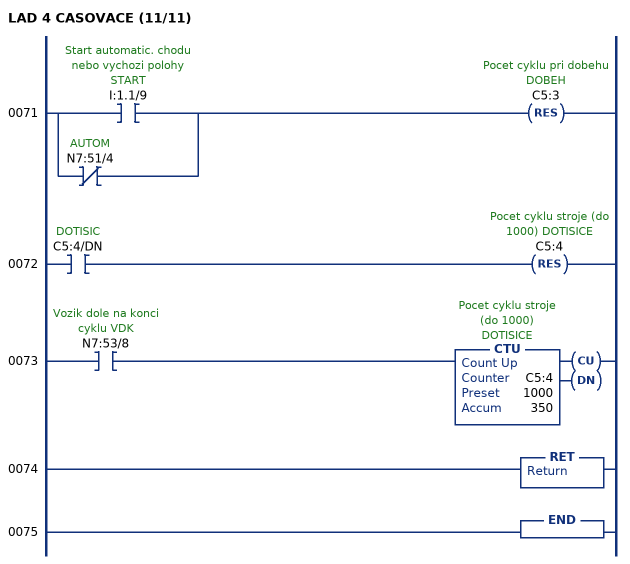
% Rung: 71 %
SOR BST XIC I:1.1/9 NXB XIO N7:51/4 BND RES C5:3 EOR
%   I:1.1/9  START  "Start automatic. chodu nebo vychozi polohy" %
%   N7:51/4  AUTOM %
%   C5:3  DOBEH  "Pocet cyklu pri dobehu" %
% Rung: 72 %
SOR XIC C5:4/DN RES C5:4 EOR
%   C5:4/DN  DOTISIC %
%   C5:4  DOTISICE  "Pocet cyklu stroje (do 1000)" %
% Rung: 73 %
SOR XIC N7:53/8 CTU C5:4 1000 350 EOR
%   N7:53/8  VDK  "Vozik dole na konci cyklu" %
%   C5:4  DOTISICE  "Pocet cyklu stroje (do 1000)" %
% Rung: 74 %
SOR RET EOR
% Rung: 75 %
SOR END EOR

LADDER 5 "DIAGN_SPOL"
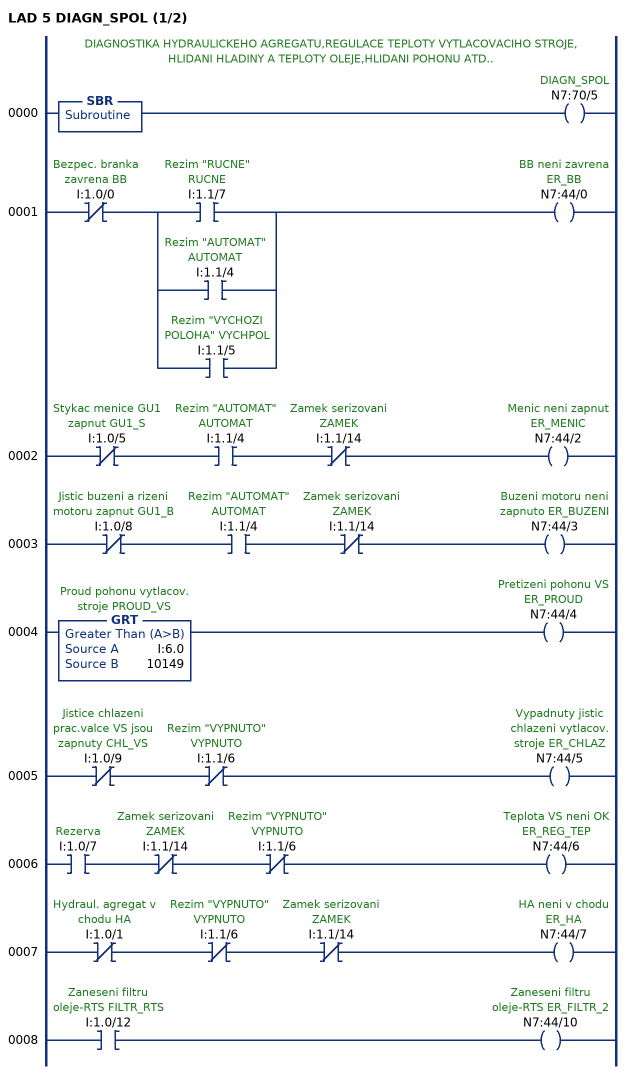
% Rung: 0 %
% DIAGNOSTIKA HYDRAULICKEHO AGREGATU,REGULACE TEPLOTY VYTLACOVACIHO STROJE,
% HLIDANI HLADINY A TEPLOTY OLEJE,HLIDANI POHONU ATD.. %
SOR SBR OTE N7:70/5 EOR
%   N7:70/5  DIAGN_SPOL %
% Rung: 1 %
SOR XIO I:1.0/0 BST XIC I:1.1/7 NXB XIC I:1.1/4 NXB XIC I:1.1/5 BND OTE N7:44/0 EOR
%   I:1.0/0  BB  "Bezpec. branka zavrena" %
%   I:1.1/7  RUCNE  "Rezim "RUCNE"" %
%   I:1.1/4  AUTOMAT  "Rezim "AUTOMAT"" %
%   I:1.1/5  VYCHPOL  "Rezim "VYCHOZI POLOHA"" %
%   N7:44/0  ER_BB  "BB neni zavrena" %
% Rung: 2 %
SOR XIO I:1.0/5 XIC I:1.1/4 XIO I:1.1/14 OTE N7:44/2 EOR
%   I:1.0/5  GU1_S  "Stykac menice GU1 zapnut" %
%   I:1.1/4  AUTOMAT  "Rezim "AUTOMAT"" %
%   I:1.1/14  ZAMEK  "Zamek serizovani" %
%   N7:44/2  ER_MENIC  "Menic neni zapnut" %
% Rung: 3 %
SOR XIO I:1.0/8 XIC I:1.1/4 XIO I:1.1/14 OTE N7:44/3 EOR
%   I:1.0/8  GU1_B  "Jistic buzeni a rizeni motoru zapnut" %
%   I:1.1/4  AUTOMAT  "Rezim "AUTOMAT"" %
%   I:1.1/14  ZAMEK  "Zamek serizovani" %
%   N7:44/3  ER_BUZENI  "Buzeni motoru neni zapnuto" %
% Rung: 4 %
SOR GRT I:6.0 10149 OTE N7:44/4 EOR
%   I:6.0  PROUD_VS  "Proud pohonu vytlacov. stroje" %
%   N7:44/4  ER_PROUD  "Pretizeni pohonu VS" %
% Rung: 5 %
SOR XIO I:1.0/9 XIO I:1.1/6 OTE N7:44/5 EOR
%   I:1.0/9  CHL_VS  "Jistice chlazeni prac.valce VS jsou zapnuty" %
%   I:1.1/6  VYPNUTO  "Rezim "VYPNUTO"" %
%   N7:44/5  ER_CHLAZ  "Vypadnuty jistic chlazeni vytlacov. stroje" %
% Rung: 6 %
SOR XIC I:1.0/7 XIO I:1.1/14 XIO I:1.1/6 OTE N7:44/6 EOR
%   I:1.0/7  "Rezerva" %
%   I:1.1/14  ZAMEK  "Zamek serizovani" %
%   I:1.1/6  VYPNUTO  "Rezim "VYPNUTO"" %
%   N7:44/6  ER_REG_TEP  "Teplota VS neni OK" %
% Rung: 7 %
SOR XIO I:1.0/1 XIO I:1.1/6 XIO I:1.1/14 OTE N7:44/7 EOR
%   I:1.0/1  HA  "Hydraul. agregat v chodu" %
%   I:1.1/6  VYPNUTO  "Rezim "VYPNUTO"" %
%   I:1.1/14  ZAMEK  "Zamek serizovani" %
%   N7:44/7  ER_HA  "HA neni v chodu" %
% Rung: 8 %
SOR XIC I:1.0/12 OTE N7:44/10 EOR
%   I:1.0/12  FILTR_RTS  "Zaneseni filtru oleje-RTS" %
%   N7:44/10  ER_FILTR_2  "Zaneseni filtru oleje-RTS" %

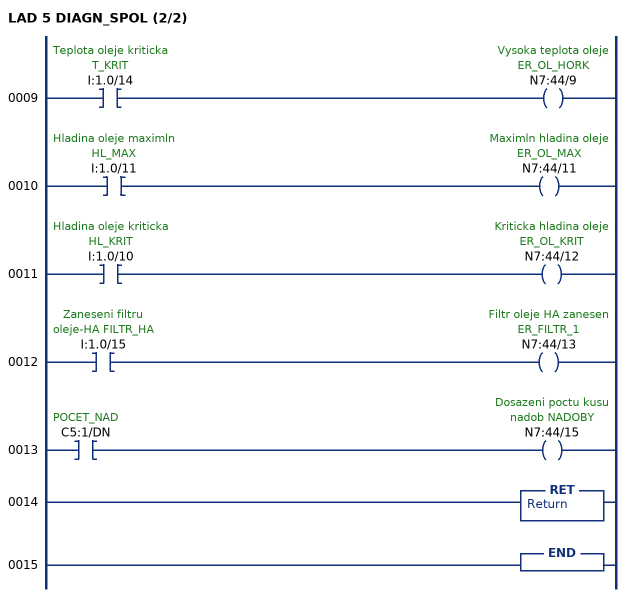
% Rung: 9 %
SOR XIC I:1.0/14 OTE N7:44/9 EOR
%   I:1.0/14  T_KRIT  "Teplota oleje kriticka" %
%   N7:44/9  ER_OL_HORK  "Vysoka teplota oleje" %
% Rung: 10 %
SOR XIC I:1.0/11 OTE N7:44/11 EOR
%   I:1.0/11  HL_MAX  "Hladina oleje maximln" %
%   N7:44/11  ER_OL_MAX  "Maximln hladina oleje" %
% Rung: 11 %
SOR XIC I:1.0/10 OTE N7:44/12 EOR
%   I:1.0/10  HL_KRIT  "Hladina oleje kriticka" %
%   N7:44/12  ER_OL_KRIT  "Kriticka hladina oleje" %
% Rung: 12 %
SOR XIC I:1.0/15 OTE N7:44/13 EOR
%   I:1.0/15  FILTR_HA  "Zaneseni filtru oleje-HA" %
%   N7:44/13  ER_FILTR_1  "Filtr oleje HA zanesen" %
% Rung: 13 %
SOR XIC C5:1/DN OTE N7:44/15 EOR
%   C5:1/DN  POCET_NAD %
%   N7:44/15  NADOBY  "Dosazeni poctu kusu nadob" %
% Rung: 14 %
SOR RET EOR
% Rung: 15 %
SOR END EOR

LADDER 6 "DIAGN_AUT"
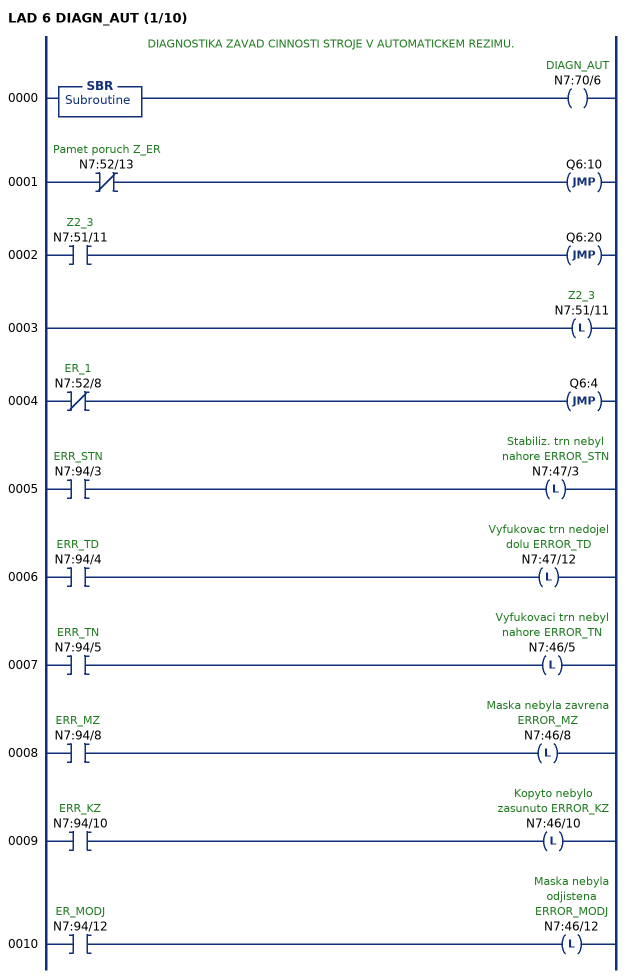
% Rung: 0 %
% DIAGNOSTIKA ZAVAD CINNOSTI STROJE V AUTOMATICKEM REZIMU. %
SOR SBR OTE N7:70/6 EOR
%   N7:70/6  DIAGN_AUT %
% Rung: 1 %
SOR XIO N7:52/13 JMP Q6:10 EOR
%   N7:52/13  Z_ER  "Pamet poruch" %
% Rung: 2 %
SOR XIC N7:51/11 JMP Q6:20 EOR
%   N7:51/11  Z2_3 %
% Rung: 3 %
SOR OTL N7:51/11 EOR
%   N7:51/11  Z2_3 %
% Rung: 4 %
SOR XIO N7:52/8 JMP Q6:4 EOR
%   N7:52/8  ER_1 %
% Rung: 5 %
SOR XIC N7:94/3 OTL N7:47/3 EOR
%   N7:94/3  ERR_STN %
%   N7:47/3  ERROR_STN  "Stabiliz. trn nebyl nahore" %
% Rung: 6 %
SOR XIC N7:94/4 OTL N7:47/12 EOR
%   N7:94/4  ERR_TD %
%   N7:47/12  ERROR_TD  "Vyfukovac trn nedojel dolu" %
% Rung: 7 %
SOR XIC N7:94/5 OTL N7:46/5 EOR
%   N7:94/5  ERR_TN %
%   N7:46/5  ERROR_TN  "Vyfukovaci trn nebyl nahore" %
% Rung: 8 %
SOR XIC N7:94/8 OTL N7:46/8 EOR
%   N7:94/8  ERR_MZ %
%   N7:46/8  ERROR_MZ  "Maska nebyla zavrena" %
% Rung: 9 %
SOR XIC N7:94/10 OTL N7:46/10 EOR
%   N7:94/10  ERR_KZ %
%   N7:46/10  ERROR_KZ  "Kopyto nebylo zasunuto" %
% Rung: 10 %
SOR XIC N7:94/12 OTL N7:46/12 EOR
%   N7:94/12  ER_MODJ %
%   N7:46/12  ERROR_MODJ  "Maska nebyla odjistena" %

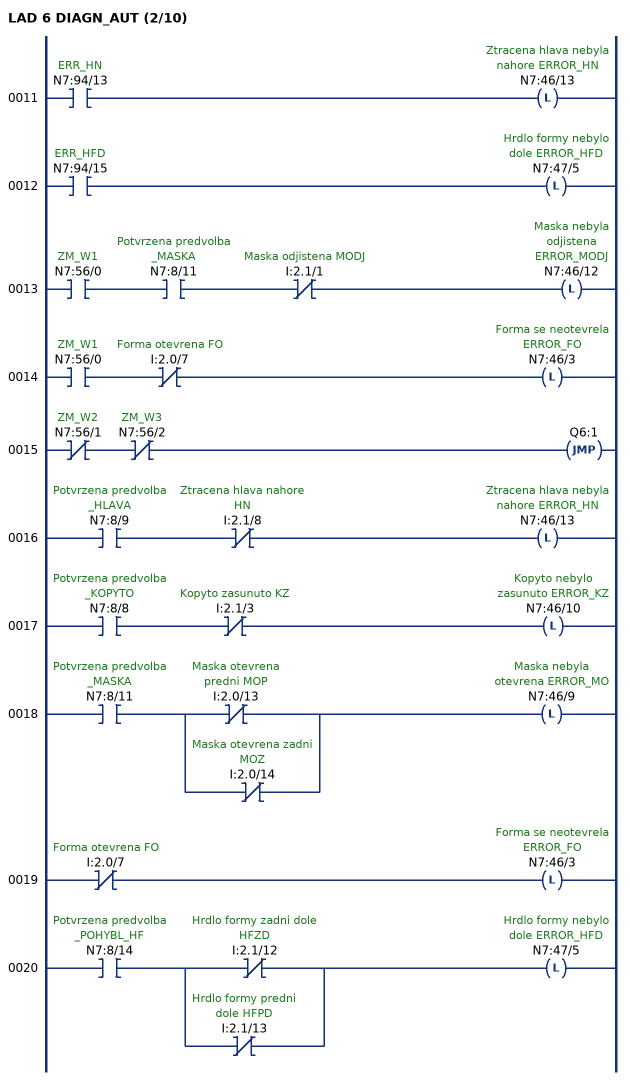
% Rung: 11 %
SOR XIC N7:94/13 OTL N7:46/13 EOR
%   N7:94/13  ERR_HN %
%   N7:46/13  ERROR_HN  "Ztracena hlava nebyla nahore" %
% Rung: 12 %
SOR XIC N7:94/15 OTL N7:47/5 EOR
%   N7:94/15  ERR_HFD %
%   N7:47/5  ERROR_HFD  "Hrdlo formy nebylo dole" %
% Rung: 13 %
SOR XIC N7:56/0 XIC N7:8/11 XIO I:2.1/1 OTL N7:46/12 EOR
%   N7:56/0  ZM_W1 %
%   N7:8/11  _MASKA  "Potvrzena predvolba" %
%   I:2.1/1  MODJ  "Maska odjistena" %
%   N7:46/12  ERROR_MODJ  "Maska nebyla odjistena" %
% Rung: 14 %
SOR XIC N7:56/0 XIO I:2.0/7 OTL N7:46/3 EOR
%   N7:56/0  ZM_W1 %
%   I:2.0/7  FO  "Forma otevrena" %
%   N7:46/3  ERROR_FO  "Forma se neotevrela" %
% Rung: 15 %
SOR XIO N7:56/1 XIO N7:56/2 JMP Q6:1 EOR
%   N7:56/1  ZM_W2 %
%   N7:56/2  ZM_W3 %
% Rung: 16 %
SOR XIC N7:8/9 XIO I:2.1/8 OTL N7:46/13 EOR
%   N7:8/9  _HLAVA  "Potvrzena predvolba" %
%   I:2.1/8  HN  "Ztracena hlava nahore" %
%   N7:46/13  ERROR_HN  "Ztracena hlava nebyla nahore" %
% Rung: 17 %
SOR XIC N7:8/8 XIO I:2.1/3 OTL N7:46/10 EOR
%   N7:8/8  _KOPYTO  "Potvrzena predvolba" %
%   I:2.1/3  KZ  "Kopyto zasunuto" %
%   N7:46/10  ERROR_KZ  "Kopyto nebylo zasunuto" %
% Rung: 18 %
SOR XIC N7:8/11 BST XIO I:2.0/13 NXB XIO I:2.0/14 BND OTL N7:46/9 EOR
%   N7:8/11  _MASKA  "Potvrzena predvolba" %
%   I:2.0/13  MOP  "Maska otevrena predni" %
%   I:2.0/14  MOZ  "Maska otevrena zadni" %
%   N7:46/9  ERROR_MO  "Maska nebyla otevrena" %
% Rung: 19 %
SOR XIO I:2.0/7 OTL N7:46/3 EOR
%   I:2.0/7  FO  "Forma otevrena" %
%   N7:46/3  ERROR_FO  "Forma se neotevrela" %
% Rung: 20 %
SOR XIC N7:8/14 BST XIO I:2.1/12 NXB XIO I:2.1/13 BND OTL N7:47/5 EOR
%   N7:8/14  _POHYBL_HF  "Potvrzena predvolba" %
%   I:2.1/12  HFZD  "Hrdlo formy zadni dole" %
%   I:2.1/13  HFPD  "Hrdlo formy predni dole" %
%   N7:47/5  ERROR_HFD  "Hrdlo formy nebylo dole" %

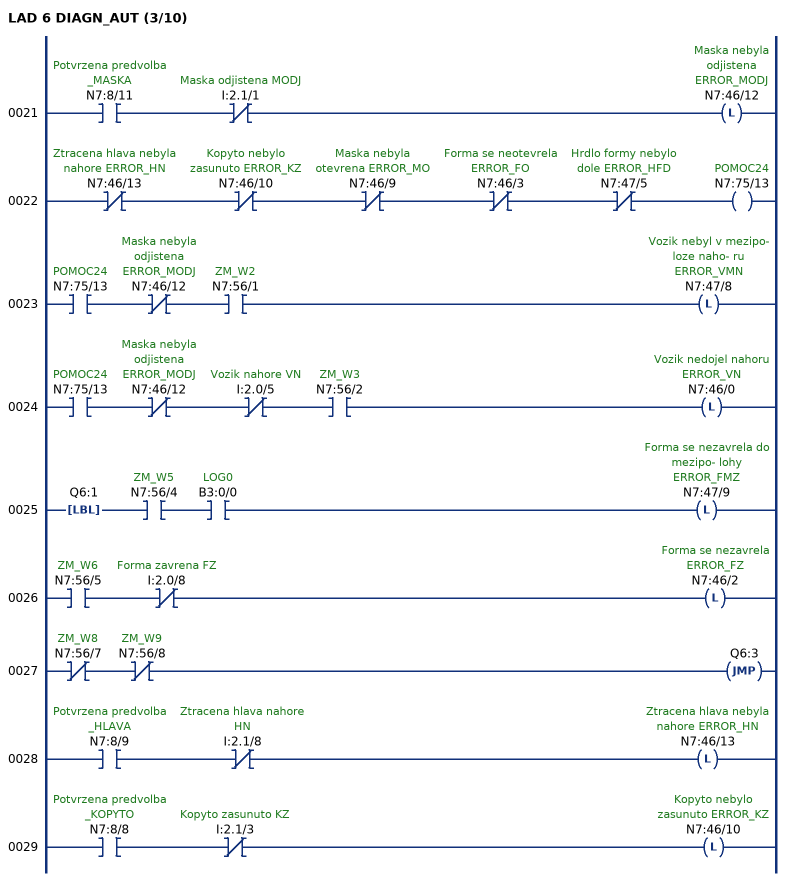
% Rung: 21 %
SOR XIC N7:8/11 XIO I:2.1/1 OTL N7:46/12 EOR
%   N7:8/11  _MASKA  "Potvrzena predvolba" %
%   I:2.1/1  MODJ  "Maska odjistena" %
%   N7:46/12  ERROR_MODJ  "Maska nebyla odjistena" %
% Rung: 22 %
SOR XIO N7:46/13 XIO N7:46/10 XIO N7:46/9 XIO N7:46/3 XIO N7:47/5 OTE N7:75/13 EOR
%   N7:46/13  ERROR_HN  "Ztracena hlava nebyla nahore" %
%   N7:46/10  ERROR_KZ  "Kopyto nebylo zasunuto" %
%   N7:46/9  ERROR_MO  "Maska nebyla otevrena" %
%   N7:46/3  ERROR_FO  "Forma se neotevrela" %
%   N7:47/5  ERROR_HFD  "Hrdlo formy nebylo dole" %
%   N7:75/13  POMOC24 %
% Rung: 23 %
SOR XIC N7:75/13 XIO N7:46/12 XIC N7:56/1 OTL N7:47/8 EOR
%   N7:75/13  POMOC24 %
%   N7:46/12  ERROR_MODJ  "Maska nebyla odjistena" %
%   N7:56/1  ZM_W2 %
%   N7:47/8  ERROR_VMN  "Vozik nebyl v mezipo- loze naho- ru" %
% Rung: 24 %
SOR XIC N7:75/13 XIO N7:46/12 XIO I:2.0/5 XIC N7:56/2 OTL N7:46/0 EOR
%   N7:75/13  POMOC24 %
%   N7:46/12  ERROR_MODJ  "Maska nebyla odjistena" %
%   I:2.0/5  VN  "Vozik nahore" %
%   N7:56/2  ZM_W3 %
%   N7:46/0  ERROR_VN  "Vozik nedojel nahoru" %
% Rung: 25 %
SOR LBL Q6:1 XIC N7:56/4 XIC B3:0/0 OTL N7:47/9 EOR
%   N7:56/4  ZM_W5 %
%   B3:0/0  LOG0 %
%   N7:47/9  ERROR_FMZ  "Forma se nezavrela do mezipo- lohy" %
% Rung: 26 %
SOR XIC N7:56/5 XIO I:2.0/8 OTL N7:46/2 EOR
%   N7:56/5  ZM_W6 %
%   I:2.0/8  FZ  "Forma zavrena" %
%   N7:46/2  ERROR_FZ  "Forma se nezavrela" %
% Rung: 27 %
SOR XIO N7:56/7 XIO N7:56/8 JMP Q6:3 EOR
%   N7:56/7  ZM_W8 %
%   N7:56/8  ZM_W9 %
% Rung: 28 %
SOR XIC N7:8/9 XIO I:2.1/8 OTL N7:46/13 EOR
%   N7:8/9  _HLAVA  "Potvrzena predvolba" %
%   I:2.1/8  HN  "Ztracena hlava nahore" %
%   N7:46/13  ERROR_HN  "Ztracena hlava nebyla nahore" %
% Rung: 29 %
SOR XIC N7:8/8 XIO I:2.1/3 OTL N7:46/10 EOR
%   N7:8/8  _KOPYTO  "Potvrzena predvolba" %
%   I:2.1/3  KZ  "Kopyto zasunuto" %
%   N7:46/10  ERROR_KZ  "Kopyto nebylo zasunuto" %

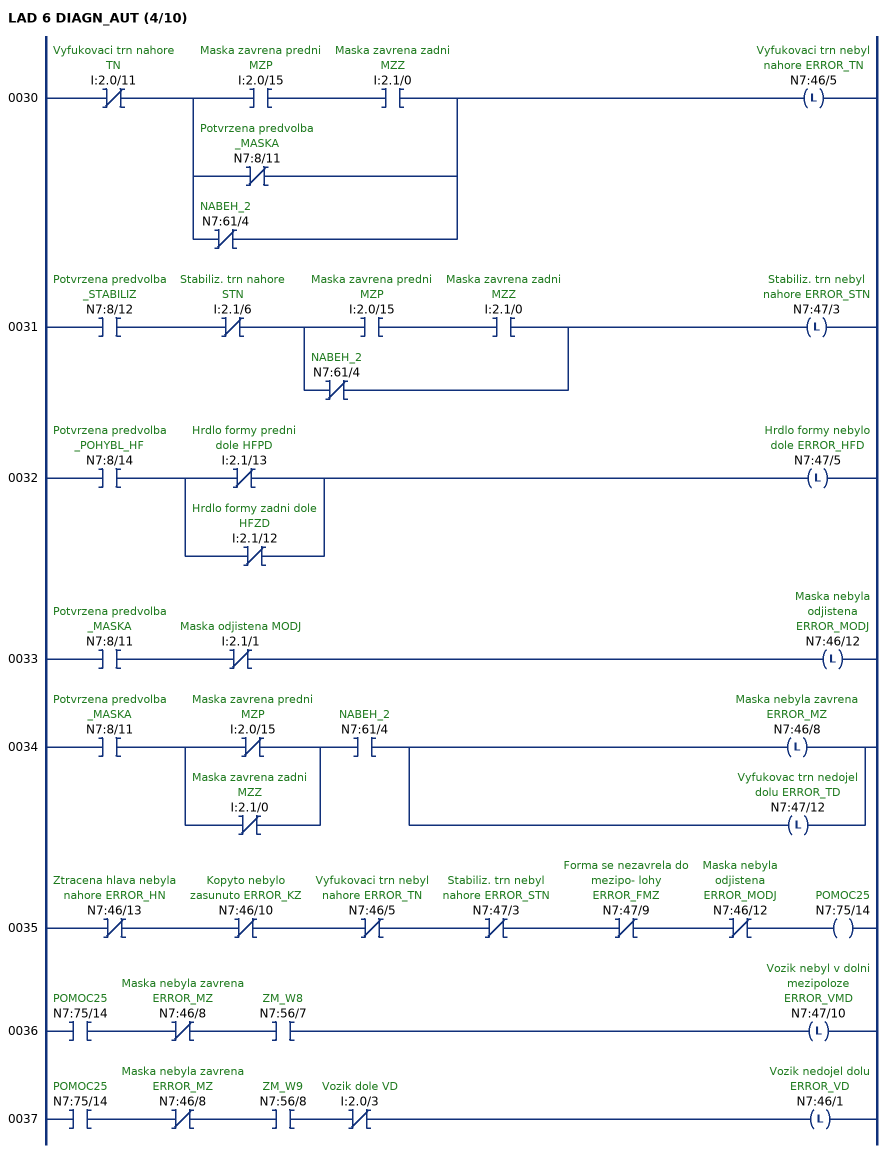
% Rung: 30 %
SOR XIO I:2.0/11 BST XIC I:2.0/15 XIC I:2.1/0 NXB XIO N7:8/11 NXB XIO N7:61/4 BND OTL N7:46/5 EOR
%   I:2.0/11  TN  "Vyfukovaci trn nahore" %
%   I:2.0/15  MZP  "Maska zavrena predni" %
%   I:2.1/0  MZZ  "Maska zavrena zadni" %
%   N7:8/11  _MASKA  "Potvrzena predvolba" %
%   N7:61/4  NABEH_2 %
%   N7:46/5  ERROR_TN  "Vyfukovaci trn nebyl nahore" %
% Rung: 31 %
SOR XIC N7:8/12 XIO I:2.1/6 BST XIC I:2.0/15 XIC I:2.1/0 NXB XIO N7:61/4 BND OTL N7:47/3 EOR
%   N7:8/12  _STABILIZ  "Potvrzena predvolba" %
%   I:2.1/6  STN  "Stabiliz. trn nahore" %
%   I:2.0/15  MZP  "Maska zavrena predni" %
%   I:2.1/0  MZZ  "Maska zavrena zadni" %
%   N7:61/4  NABEH_2 %
%   N7:47/3  ERROR_STN  "Stabiliz. trn nebyl nahore" %
% Rung: 32 %
SOR XIC N7:8/14 BST XIO I:2.1/13 NXB XIO I:2.1/12 BND OTL N7:47/5 EOR
%   N7:8/14  _POHYBL_HF  "Potvrzena predvolba" %
%   I:2.1/13  HFPD  "Hrdlo formy predni dole" %
%   I:2.1/12  HFZD  "Hrdlo formy zadni dole" %
%   N7:47/5  ERROR_HFD  "Hrdlo formy nebylo dole" %
% Rung: 33 %
SOR XIC N7:8/11 XIO I:2.1/1 OTL N7:46/12 EOR
%   N7:8/11  _MASKA  "Potvrzena predvolba" %
%   I:2.1/1  MODJ  "Maska odjistena" %
%   N7:46/12  ERROR_MODJ  "Maska nebyla odjistena" %
% Rung: 34 %
SOR XIC N7:8/11 BST XIO I:2.0/15 NXB XIO I:2.1/0 BND XIC N7:61/4 BST OTL N7:46/8 NXB OTL N7:47/12 BND EOR
%   N7:8/11  _MASKA  "Potvrzena predvolba" %
%   I:2.0/15  MZP  "Maska zavrena predni" %
%   I:2.1/0  MZZ  "Maska zavrena zadni" %
%   N7:61/4  NABEH_2 %
%   N7:46/8  ERROR_MZ  "Maska nebyla zavrena" %
%   N7:47/12  ERROR_TD  "Vyfukovac trn nedojel dolu" %
% Rung: 35 %
SOR XIO N7:46/13 XIO N7:46/10 XIO N7:46/5 XIO N7:47/3 XIO N7:47/9 XIO N7:46/12 OTE N7:75/14 EOR
%   N7:46/13  ERROR_HN  "Ztracena hlava nebyla nahore" %
%   N7:46/10  ERROR_KZ  "Kopyto nebylo zasunuto" %
%   N7:46/5  ERROR_TN  "Vyfukovaci trn nebyl nahore" %
%   N7:47/3  ERROR_STN  "Stabiliz. trn nebyl nahore" %
%   N7:47/9  ERROR_FMZ  "Forma se nezavrela do mezipo- lohy" %
%   N7:46/12  ERROR_MODJ  "Maska nebyla odjistena" %
%   N7:75/14  POMOC25 %
% Rung: 36 %
SOR XIC N7:75/14 XIO N7:46/8 XIC N7:56/7 OTL N7:47/10 EOR
%   N7:75/14  POMOC25 %
%   N7:46/8  ERROR_MZ  "Maska nebyla zavrena" %
%   N7:56/7  ZM_W8 %
%   N7:47/10  ERROR_VMD  "Vozik nebyl v dolni mezipoloze" %
% Rung: 37 %
SOR XIC N7:75/14 XIO N7:46/8 XIC N7:56/8 XIO I:2.0/3 OTL N7:46/1 EOR
%   N7:75/14  POMOC25 %
%   N7:46/8  ERROR_MZ  "Maska nebyla zavrena" %
%   N7:56/8  ZM_W9 %
%   I:2.0/3  VD  "Vozik dole" %
%   N7:46/1  ERROR_VD  "Vozik nedojel dolu" %

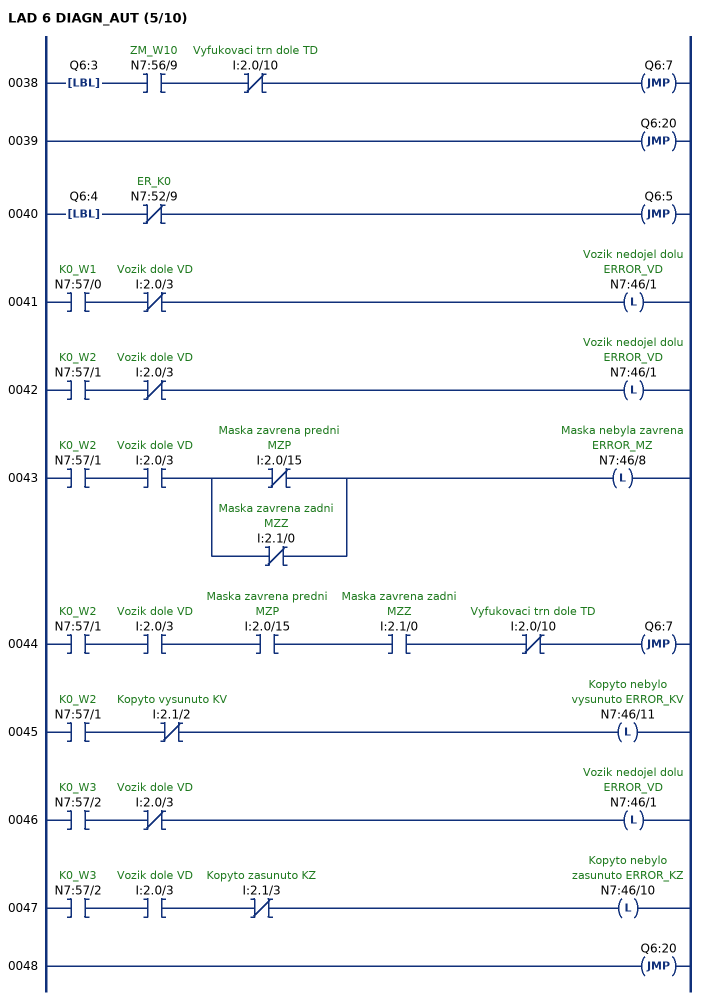
% Rung: 38 %
SOR LBL Q6:3 XIC N7:56/9 XIO I:2.0/10 JMP Q6:7 EOR
%   N7:56/9  ZM_W10 %
%   I:2.0/10  TD  "Vyfukovaci trn dole" %
% Rung: 39 %
SOR JMP Q6:20 EOR
% Rung: 40 %
SOR LBL Q6:4 XIO N7:52/9 JMP Q6:5 EOR
%   N7:52/9  ER_K0 %
% Rung: 41 %
SOR XIC N7:57/0 XIO I:2.0/3 OTL N7:46/1 EOR
%   N7:57/0  K0_W1 %
%   I:2.0/3  VD  "Vozik dole" %
%   N7:46/1  ERROR_VD  "Vozik nedojel dolu" %
% Rung: 42 %
SOR XIC N7:57/1 XIO I:2.0/3 OTL N7:46/1 EOR
%   N7:57/1  K0_W2 %
%   I:2.0/3  VD  "Vozik dole" %
%   N7:46/1  ERROR_VD  "Vozik nedojel dolu" %
% Rung: 43 %
SOR XIC N7:57/1 XIC I:2.0/3 BST XIO I:2.0/15 NXB XIO I:2.1/0 BND OTL N7:46/8 EOR
%   N7:57/1  K0_W2 %
%   I:2.0/3  VD  "Vozik dole" %
%   I:2.0/15  MZP  "Maska zavrena predni" %
%   I:2.1/0  MZZ  "Maska zavrena zadni" %
%   N7:46/8  ERROR_MZ  "Maska nebyla zavrena" %
% Rung: 44 %
SOR XIC N7:57/1 XIC I:2.0/3 XIC I:2.0/15 XIC I:2.1/0 XIO I:2.0/10 JMP Q6:7 EOR
%   N7:57/1  K0_W2 %
%   I:2.0/3  VD  "Vozik dole" %
%   I:2.0/15  MZP  "Maska zavrena predni" %
%   I:2.1/0  MZZ  "Maska zavrena zadni" %
%   I:2.0/10  TD  "Vyfukovaci trn dole" %
% Rung: 45 %
SOR XIC N7:57/1 XIO I:2.1/2 OTL N7:46/11 EOR
%   N7:57/1  K0_W2 %
%   I:2.1/2  KV  "Kopyto vysunuto" %
%   N7:46/11  ERROR_KV  "Kopyto nebylo vysunuto" %
% Rung: 46 %
SOR XIC N7:57/2 XIO I:2.0/3 OTL N7:46/1 EOR
%   N7:57/2  K0_W3 %
%   I:2.0/3  VD  "Vozik dole" %
%   N7:46/1  ERROR_VD  "Vozik nedojel dolu" %
% Rung: 47 %
SOR XIC N7:57/2 XIC I:2.0/3 XIO I:2.1/3 OTL N7:46/10 EOR
%   N7:57/2  K0_W3 %
%   I:2.0/3  VD  "Vozik dole" %
%   I:2.1/3  KZ  "Kopyto zasunuto" %
%   N7:46/10  ERROR_KZ  "Kopyto nebylo zasunuto" %
% Rung: 48 %
SOR JMP Q6:20 EOR

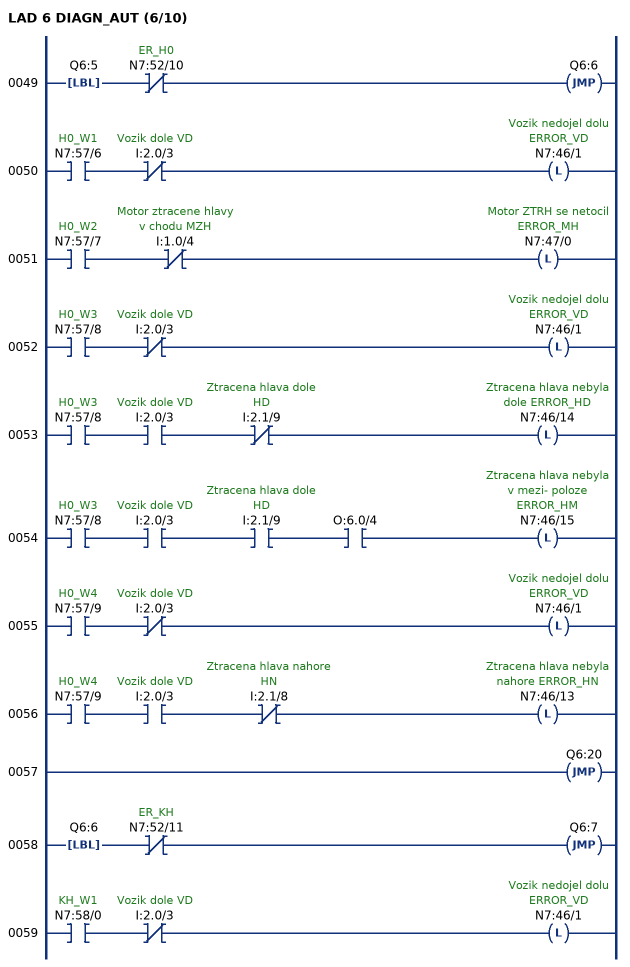
% Rung: 49 %
SOR LBL Q6:5 XIO N7:52/10 JMP Q6:6 EOR
%   N7:52/10  ER_H0 %
% Rung: 50 %
SOR XIC N7:57/6 XIO I:2.0/3 OTL N7:46/1 EOR
%   N7:57/6  H0_W1 %
%   I:2.0/3  VD  "Vozik dole" %
%   N7:46/1  ERROR_VD  "Vozik nedojel dolu" %
% Rung: 51 %
SOR XIC N7:57/7 XIO I:1.0/4 OTL N7:47/0 EOR
%   N7:57/7  H0_W2 %
%   I:1.0/4  MZH  "Motor ztracene hlavy v chodu" %
%   N7:47/0  ERROR_MH  "Motor ZTRH se netocil" %
% Rung: 52 %
SOR XIC N7:57/8 XIO I:2.0/3 OTL N7:46/1 EOR
%   N7:57/8  H0_W3 %
%   I:2.0/3  VD  "Vozik dole" %
%   N7:46/1  ERROR_VD  "Vozik nedojel dolu" %
% Rung: 53 %
SOR XIC N7:57/8 XIC I:2.0/3 XIO I:2.1/9 OTL N7:46/14 EOR
%   N7:57/8  H0_W3 %
%   I:2.0/3  VD  "Vozik dole" %
%   I:2.1/9  HD  "Ztracena hlava dole" %
%   N7:46/14  ERROR_HD  "Ztracena hlava nebyla dole" %
% Rung: 54 %
SOR XIC N7:57/8 XIC I:2.0/3 XIC I:2.1/9 XIC O:6.0/4 OTL N7:46/15 EOR
%   N7:57/8  H0_W3 %
%   I:2.0/3  VD  "Vozik dole" %
%   I:2.1/9  HD  "Ztracena hlava dole" %
%   N7:46/15  ERROR_HM  "Ztracena hlava nebyla v mezi- poloze" %
% Rung: 55 %
SOR XIC N7:57/9 XIO I:2.0/3 OTL N7:46/1 EOR
%   N7:57/9  H0_W4 %
%   I:2.0/3  VD  "Vozik dole" %
%   N7:46/1  ERROR_VD  "Vozik nedojel dolu" %
% Rung: 56 %
SOR XIC N7:57/9 XIC I:2.0/3 XIO I:2.1/8 OTL N7:46/13 EOR
%   N7:57/9  H0_W4 %
%   I:2.0/3  VD  "Vozik dole" %
%   I:2.1/8  HN  "Ztracena hlava nahore" %
%   N7:46/13  ERROR_HN  "Ztracena hlava nebyla nahore" %
% Rung: 57 %
SOR JMP Q6:20 EOR
% Rung: 58 %
SOR LBL Q6:6 XIO N7:52/11 JMP Q6:7 EOR
%   N7:52/11  ER_KH %
% Rung: 59 %
SOR XIC N7:58/0 XIO I:2.0/3 OTL N7:46/1 EOR
%   N7:58/0  KH_W1 %
%   I:2.0/3  VD  "Vozik dole" %
%   N7:46/1  ERROR_VD  "Vozik nedojel dolu" %

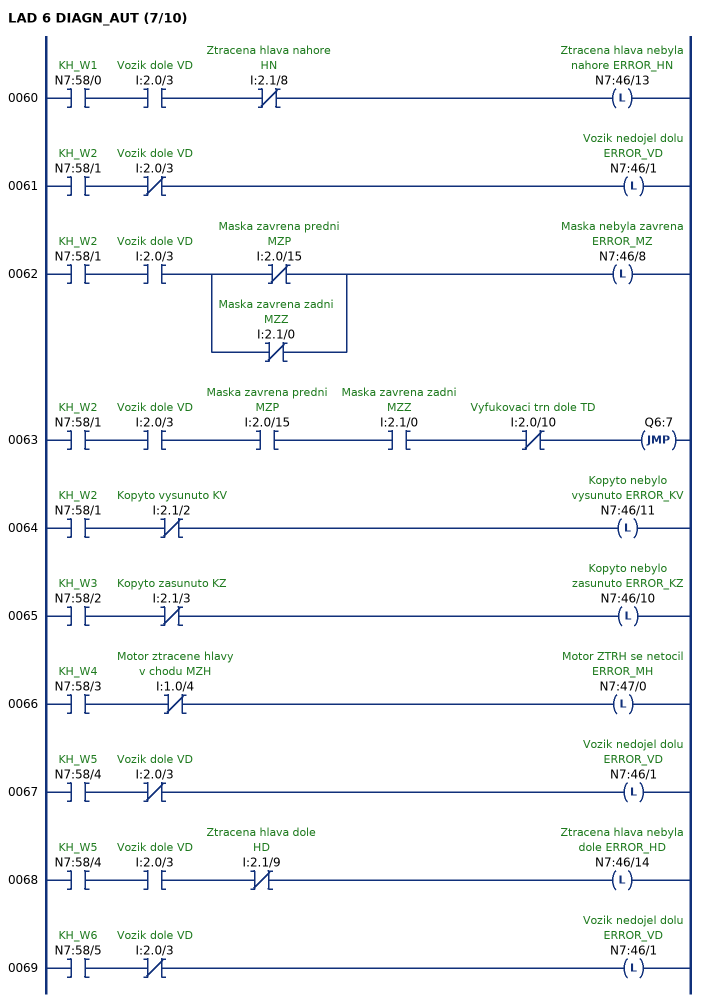
% Rung: 60 %
SOR XIC N7:58/0 XIC I:2.0/3 XIO I:2.1/8 OTL N7:46/13 EOR
%   N7:58/0  KH_W1 %
%   I:2.0/3  VD  "Vozik dole" %
%   I:2.1/8  HN  "Ztracena hlava nahore" %
%   N7:46/13  ERROR_HN  "Ztracena hlava nebyla nahore" %
% Rung: 61 %
SOR XIC N7:58/1 XIO I:2.0/3 OTL N7:46/1 EOR
%   N7:58/1  KH_W2 %
%   I:2.0/3  VD  "Vozik dole" %
%   N7:46/1  ERROR_VD  "Vozik nedojel dolu" %
% Rung: 62 %
SOR XIC N7:58/1 XIC I:2.0/3 BST XIO I:2.0/15 NXB XIO I:2.1/0 BND OTL N7:46/8 EOR
%   N7:58/1  KH_W2 %
%   I:2.0/3  VD  "Vozik dole" %
%   I:2.0/15  MZP  "Maska zavrena predni" %
%   I:2.1/0  MZZ  "Maska zavrena zadni" %
%   N7:46/8  ERROR_MZ  "Maska nebyla zavrena" %
% Rung: 63 %
SOR XIC N7:58/1 XIC I:2.0/3 XIC I:2.0/15 XIC I:2.1/0 XIO I:2.0/10 JMP Q6:7 EOR
%   N7:58/1  KH_W2 %
%   I:2.0/3  VD  "Vozik dole" %
%   I:2.0/15  MZP  "Maska zavrena predni" %
%   I:2.1/0  MZZ  "Maska zavrena zadni" %
%   I:2.0/10  TD  "Vyfukovaci trn dole" %
% Rung: 64 %
SOR XIC N7:58/1 XIO I:2.1/2 OTL N7:46/11 EOR
%   N7:58/1  KH_W2 %
%   I:2.1/2  KV  "Kopyto vysunuto" %
%   N7:46/11  ERROR_KV  "Kopyto nebylo vysunuto" %
% Rung: 65 %
SOR XIC N7:58/2 XIO I:2.1/3 OTL N7:46/10 EOR
%   N7:58/2  KH_W3 %
%   I:2.1/3  KZ  "Kopyto zasunuto" %
%   N7:46/10  ERROR_KZ  "Kopyto nebylo zasunuto" %
% Rung: 66 %
SOR XIC N7:58/3 XIO I:1.0/4 OTL N7:47/0 EOR
%   N7:58/3  KH_W4 %
%   I:1.0/4  MZH  "Motor ztracene hlavy v chodu" %
%   N7:47/0  ERROR_MH  "Motor ZTRH se netocil" %
% Rung: 67 %
SOR XIC N7:58/4 XIO I:2.0/3 OTL N7:46/1 EOR
%   N7:58/4  KH_W5 %
%   I:2.0/3  VD  "Vozik dole" %
%   N7:46/1  ERROR_VD  "Vozik nedojel dolu" %
% Rung: 68 %
SOR XIC N7:58/4 XIC I:2.0/3 XIO I:2.1/9 OTL N7:46/14 EOR
%   N7:58/4  KH_W5 %
%   I:2.0/3  VD  "Vozik dole" %
%   I:2.1/9  HD  "Ztracena hlava dole" %
%   N7:46/14  ERROR_HD  "Ztracena hlava nebyla dole" %
% Rung: 69 %
SOR XIC N7:58/5 XIO I:2.0/3 OTL N7:46/1 EOR
%   N7:58/5  KH_W6 %
%   I:2.0/3  VD  "Vozik dole" %
%   N7:46/1  ERROR_VD  "Vozik nedojel dolu" %

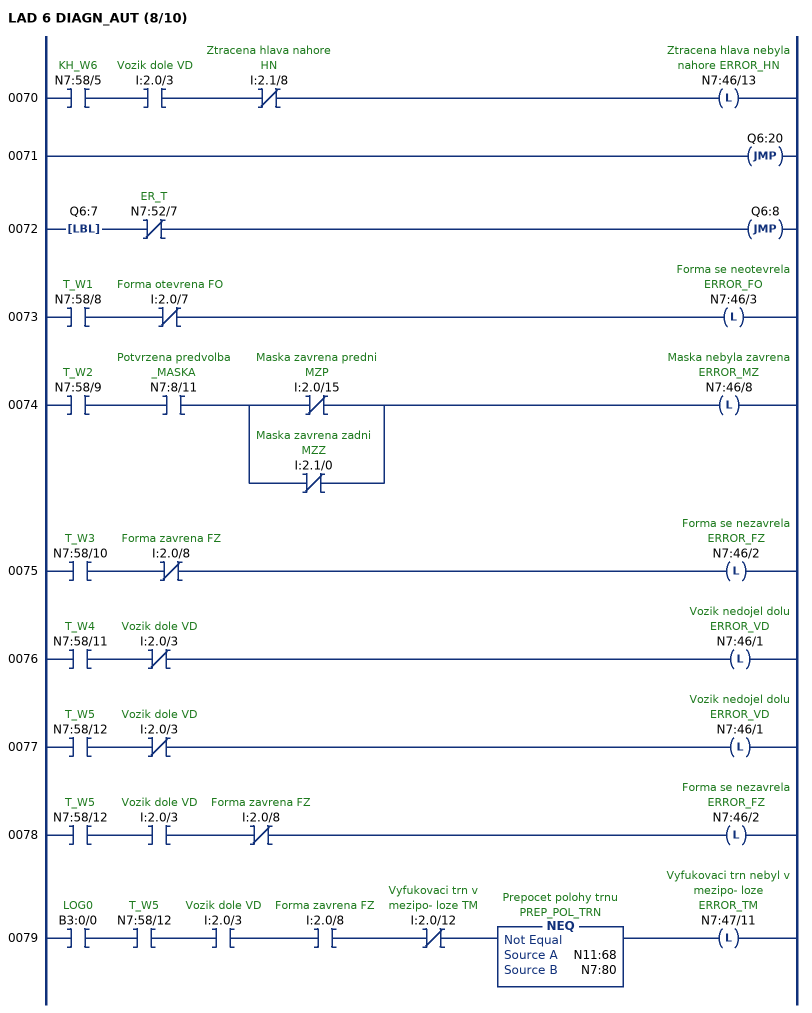
% Rung: 70 %
SOR XIC N7:58/5 XIC I:2.0/3 XIO I:2.1/8 OTL N7:46/13 EOR
%   N7:58/5  KH_W6 %
%   I:2.0/3  VD  "Vozik dole" %
%   I:2.1/8  HN  "Ztracena hlava nahore" %
%   N7:46/13  ERROR_HN  "Ztracena hlava nebyla nahore" %
% Rung: 71 %
SOR JMP Q6:20 EOR
% Rung: 72 %
SOR LBL Q6:7 XIO N7:52/7 JMP Q6:8 EOR
%   N7:52/7  ER_T %
% Rung: 73 %
SOR XIC N7:58/8 XIO I:2.0/7 OTL N7:46/3 EOR
%   N7:58/8  T_W1 %
%   I:2.0/7  FO  "Forma otevrena" %
%   N7:46/3  ERROR_FO  "Forma se neotevrela" %
% Rung: 74 %
SOR XIC N7:58/9 XIC N7:8/11 BST XIO I:2.0/15 NXB XIO I:2.1/0 BND OTL N7:46/8 EOR
%   N7:58/9  T_W2 %
%   N7:8/11  _MASKA  "Potvrzena predvolba" %
%   I:2.0/15  MZP  "Maska zavrena predni" %
%   I:2.1/0  MZZ  "Maska zavrena zadni" %
%   N7:46/8  ERROR_MZ  "Maska nebyla zavrena" %
% Rung: 75 %
SOR XIC N7:58/10 XIO I:2.0/8 OTL N7:46/2 EOR
%   N7:58/10  T_W3 %
%   I:2.0/8  FZ  "Forma zavrena" %
%   N7:46/2  ERROR_FZ  "Forma se nezavrela" %
% Rung: 76 %
SOR XIC N7:58/11 XIO I:2.0/3 OTL N7:46/1 EOR
%   N7:58/11  T_W4 %
%   I:2.0/3  VD  "Vozik dole" %
%   N7:46/1  ERROR_VD  "Vozik nedojel dolu" %
% Rung: 77 %
SOR XIC N7:58/12 XIO I:2.0/3 OTL N7:46/1 EOR
%   N7:58/12  T_W5 %
%   I:2.0/3  VD  "Vozik dole" %
%   N7:46/1  ERROR_VD  "Vozik nedojel dolu" %
% Rung: 78 %
SOR XIC N7:58/12 XIC I:2.0/3 XIO I:2.0/8 OTL N7:46/2 EOR
%   N7:58/12  T_W5 %
%   I:2.0/3  VD  "Vozik dole" %
%   I:2.0/8  FZ  "Forma zavrena" %
%   N7:46/2  ERROR_FZ  "Forma se nezavrela" %
% Rung: 79 %
SOR XIC B3:0/0 XIC N7:58/12 XIC I:2.0/3 XIC I:2.0/8 XIO I:2.0/12 NEQ N11:68 N7:80 OTL N7:47/11 EOR
%   B3:0/0  LOG0 %
%   N7:58/12  T_W5 %
%   I:2.0/3  VD  "Vozik dole" %
%   I:2.0/8  FZ  "Forma zavrena" %
%   I:2.0/12  TM  "Vyfukovaci trn v mezipo- loze" %
%   N11:68  PREP_POL_TRN  "Prepocet polohy trnu" %
%   N7:47/11  ERROR_TM  "Vyfukovaci trn nebyl v mezipo- loze" %

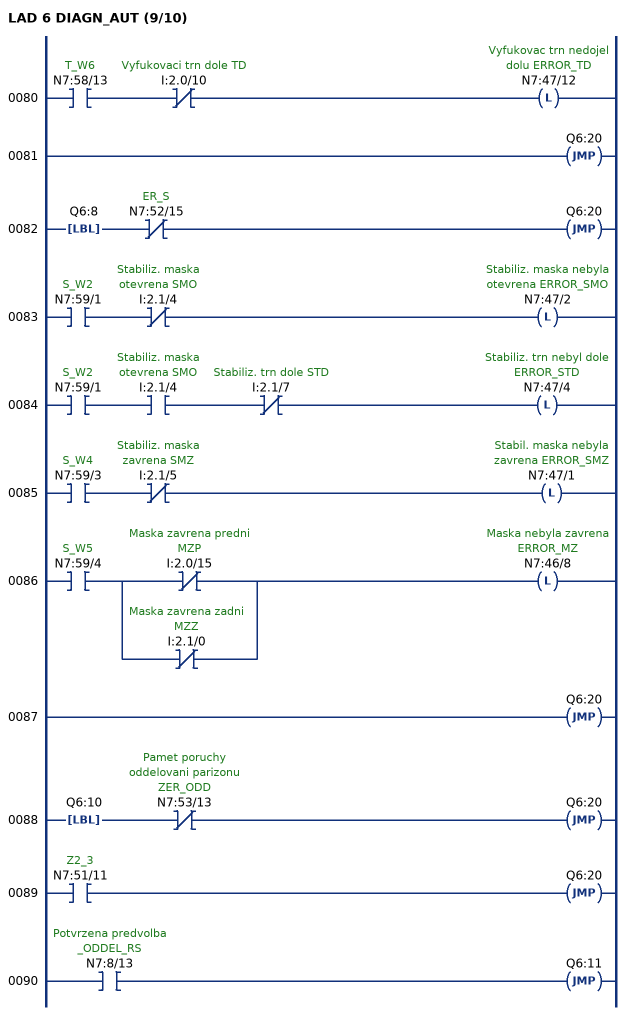
% Rung: 80 %
SOR XIC N7:58/13 XIO I:2.0/10 OTL N7:47/12 EOR
%   N7:58/13  T_W6 %
%   I:2.0/10  TD  "Vyfukovaci trn dole" %
%   N7:47/12  ERROR_TD  "Vyfukovac trn nedojel dolu" %
% Rung: 81 %
SOR JMP Q6:20 EOR
% Rung: 82 %
SOR LBL Q6:8 XIO N7:52/15 JMP Q6:20 EOR
%   N7:52/15  ER_S %
% Rung: 83 %
SOR XIC N7:59/1 XIO I:2.1/4 OTL N7:47/2 EOR
%   N7:59/1  S_W2 %
%   I:2.1/4  SMO  "Stabiliz. maska otevrena" %
%   N7:47/2  ERROR_SMO  "Stabiliz. maska nebyla otevrena" %
% Rung: 84 %
SOR XIC N7:59/1 XIC I:2.1/4 XIO I:2.1/7 OTL N7:47/4 EOR
%   N7:59/1  S_W2 %
%   I:2.1/4  SMO  "Stabiliz. maska otevrena" %
%   I:2.1/7  STD  "Stabiliz. trn dole" %
%   N7:47/4  ERROR_STD  "Stabiliz. trn nebyl dole" %
% Rung: 85 %
SOR XIC N7:59/3 XIO I:2.1/5 OTL N7:47/1 EOR
%   N7:59/3  S_W4 %
%   I:2.1/5  SMZ  "Stabiliz. maska zavrena" %
%   N7:47/1  ERROR_SMZ  "Stabil. maska nebyla zavrena" %
% Rung: 86 %
SOR XIC N7:59/4 BST XIO I:2.0/15 NXB XIO I:2.1/0 BND OTL N7:46/8 EOR
%   N7:59/4  S_W5 %
%   I:2.0/15  MZP  "Maska zavrena predni" %
%   I:2.1/0  MZZ  "Maska zavrena zadni" %
%   N7:46/8  ERROR_MZ  "Maska nebyla zavrena" %
% Rung: 87 %
SOR JMP Q6:20 EOR
% Rung: 88 %
SOR LBL Q6:10 XIO N7:53/13 JMP Q6:20 EOR
%   N7:53/13  ZER_ODD  "Pamet poruchy oddelovani parizonu" %
% Rung: 89 %
SOR XIC N7:51/11 JMP Q6:20 EOR
%   N7:51/11  Z2_3 %
% Rung: 90 %
SOR XIC N7:8/13 JMP Q6:11 EOR
%   N7:8/13  _ODDEL_RS  "Potvrzena predvolba" %

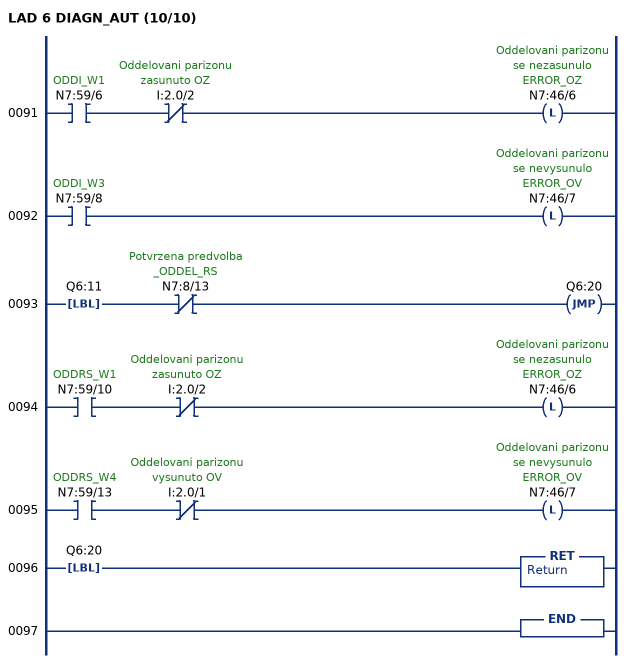
% Rung: 91 %
SOR XIC N7:59/6 XIO I:2.0/2 OTL N7:46/6 EOR
%   N7:59/6  ODDI_W1 %
%   I:2.0/2  OZ  "Oddelovani parizonu zasunuto" %
%   N7:46/6  ERROR_OZ  "Oddelovani parizonu se nezasunulo" %
% Rung: 92 %
SOR XIC N7:59/8 OTL N7:46/7 EOR
%   N7:59/8  ODDI_W3 %
%   N7:46/7  ERROR_OV  "Oddelovani parizonu se nevysunulo" %
% Rung: 93 %
SOR LBL Q6:11 XIO N7:8/13 JMP Q6:20 EOR
%   N7:8/13  _ODDEL_RS  "Potvrzena predvolba" %
% Rung: 94 %
SOR XIC N7:59/10 XIO I:2.0/2 OTL N7:46/6 EOR
%   N7:59/10  ODDRS_W1 %
%   I:2.0/2  OZ  "Oddelovani parizonu zasunuto" %
%   N7:46/6  ERROR_OZ  "Oddelovani parizonu se nezasunulo" %
% Rung: 95 %
SOR XIC N7:59/13 XIO I:2.0/1 OTL N7:46/7 EOR
%   N7:59/13  ODDRS_W4 %
%   I:2.0/1  OV  "Oddelovani parizonu vysunuto" %
%   N7:46/7  ERROR_OV  "Oddelovani parizonu se nevysunulo" %
% Rung: 96 %
SOR LBL Q6:20 RET EOR
% Rung: 97 %
SOR END EOR

LADDER 7 "DIAGN_K_VP"
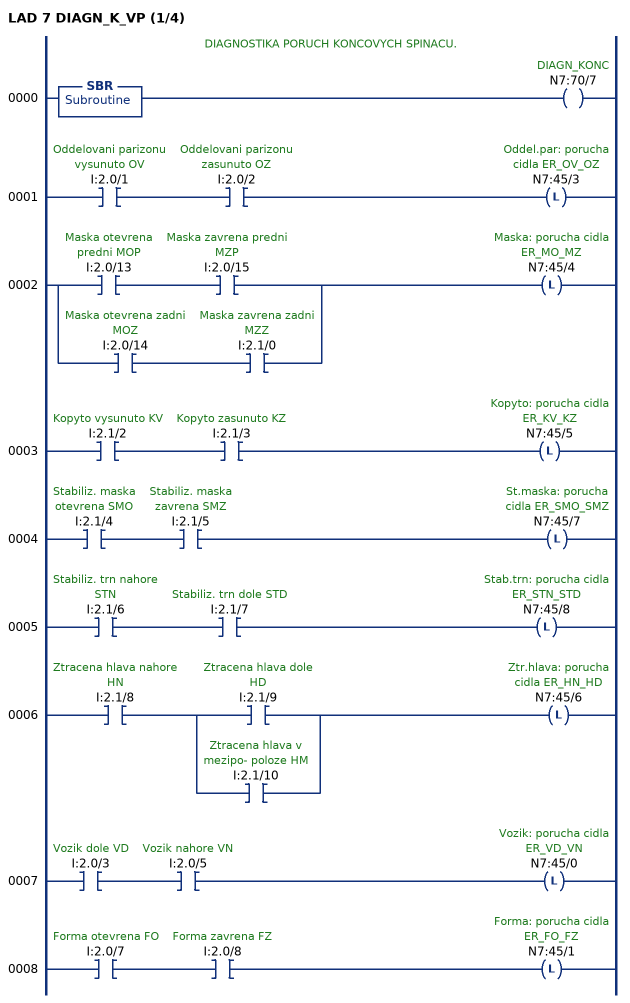
% Rung: 0 %
% DIAGNOSTIKA PORUCH KONCOVYCH SPINACU. %
SOR SBR OTE N7:70/7 EOR
%   N7:70/7  DIAGN_KONC %
% Rung: 1 %
SOR XIC I:2.0/1 XIC I:2.0/2 OTL N7:45/3 EOR
%   I:2.0/1  OV  "Oddelovani parizonu vysunuto" %
%   I:2.0/2  OZ  "Oddelovani parizonu zasunuto" %
%   N7:45/3  ER_OV_OZ  "Oddel.par: porucha cidla" %
% Rung: 2 %
SOR BST XIC I:2.0/13 XIC I:2.0/15 NXB XIC I:2.0/14 XIC I:2.1/0 BND OTL N7:45/4 EOR
%   I:2.0/13  MOP  "Maska otevrena predni" %
%   I:2.0/15  MZP  "Maska zavrena predni" %
%   I:2.0/14  MOZ  "Maska otevrena zadni" %
%   I:2.1/0  MZZ  "Maska zavrena zadni" %
%   N7:45/4  ER_MO_MZ  "Maska: porucha cidla" %
% Rung: 3 %
SOR XIC I:2.1/2 XIC I:2.1/3 OTL N7:45/5 EOR
%   I:2.1/2  KV  "Kopyto vysunuto" %
%   I:2.1/3  KZ  "Kopyto zasunuto" %
%   N7:45/5  ER_KV_KZ  "Kopyto: porucha cidla" %
% Rung: 4 %
SOR XIC I:2.1/4 XIC I:2.1/5 OTL N7:45/7 EOR
%   I:2.1/4  SMO  "Stabiliz. maska otevrena" %
%   I:2.1/5  SMZ  "Stabiliz. maska zavrena" %
%   N7:45/7  ER_SMO_SMZ  "St.maska: porucha cidla" %
% Rung: 5 %
SOR XIC I:2.1/6 XIC I:2.1/7 OTL N7:45/8 EOR
%   I:2.1/6  STN  "Stabiliz. trn nahore" %
%   I:2.1/7  STD  "Stabiliz. trn dole" %
%   N7:45/8  ER_STN_STD  "Stab.trn: porucha cidla" %
% Rung: 6 %
SOR XIC I:2.1/8 BST XIC I:2.1/9 NXB XIC I:2.1/10 BND OTL N7:45/6 EOR
%   I:2.1/8  HN  "Ztracena hlava nahore" %
%   I:2.1/9  HD  "Ztracena hlava dole" %
%   I:2.1/10  HM  "Ztracena hlava v mezipo- poloze" %
%   N7:45/6  ER_HN_HD  "Ztr.hlava: porucha cidla" %
% Rung: 7 %
SOR XIC I:2.0/3 XIC I:2.0/5 OTL N7:45/0 EOR
%   I:2.0/3  VD  "Vozik dole" %
%   I:2.0/5  VN  "Vozik nahore" %
%   N7:45/0  ER_VD_VN  "Vozik: porucha cidla" %
% Rung: 8 %
SOR XIC I:2.0/7 XIC I:2.0/8 OTL N7:45/1 EOR
%   I:2.0/7  FO  "Forma otevrena" %
%   I:2.0/8  FZ  "Forma zavrena" %
%   N7:45/1  ER_FO_FZ  "Forma: porucha cidla" %

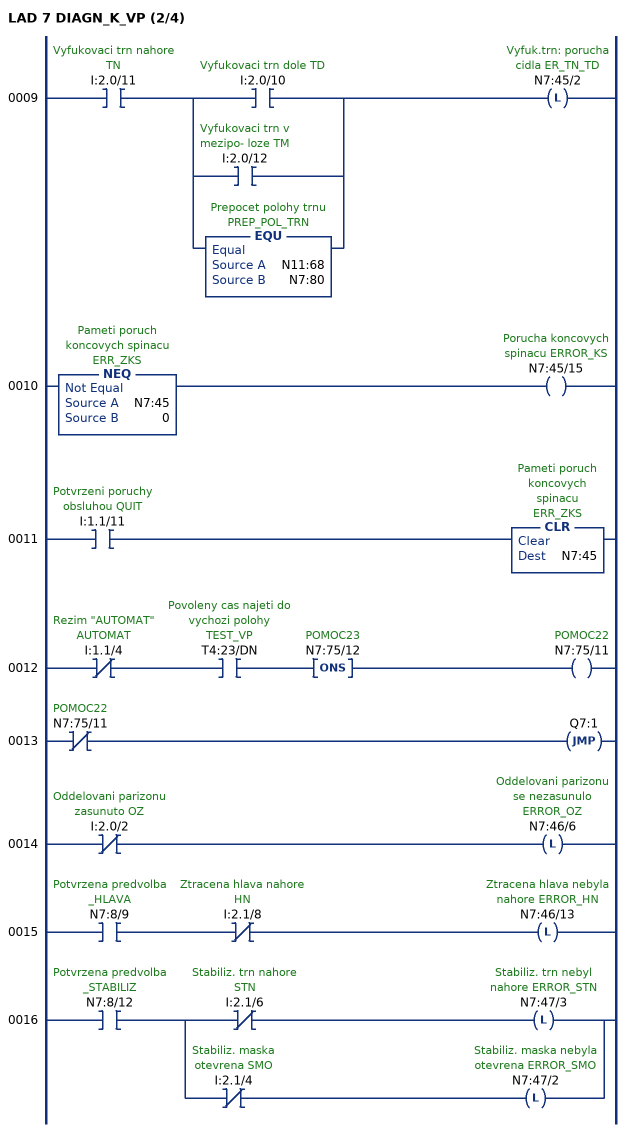
% Rung: 9 %
SOR XIC I:2.0/11 BST XIC I:2.0/10 NXB XIC I:2.0/12 NXB EQU N11:68 N7:80 BND OTL N7:45/2 EOR
%   I:2.0/11  TN  "Vyfukovaci trn nahore" %
%   I:2.0/10  TD  "Vyfukovaci trn dole" %
%   I:2.0/12  TM  "Vyfukovaci trn v mezipo- loze" %
%   N11:68  PREP_POL_TRN  "Prepocet polohy trnu" %
%   N7:45/2  ER_TN_TD  "Vyfuk.trn: porucha cidla" %
% Rung: 10 %
SOR NEQ N7:45 0 OTE N7:45/15 EOR
%   N7:45  ERR_ZKS  "Pameti poruch koncovych spinacu" %
%   N7:45/15  ERROR_KS  "Porucha koncovych spinacu" %
% Rung: 11 %
SOR XIC I:1.1/11 CLR N7:45 EOR
%   I:1.1/11  QUIT  "Potvrzeni poruchy obsluhou" %
%   N7:45  ERR_ZKS  "Pameti poruch koncovych spinacu" %
% Rung: 12 %
SOR XIO I:1.1/4 XIC T4:23/DN OSR N7:75/12 OTE N7:75/11 EOR
%   I:1.1/4  AUTOMAT  "Rezim "AUTOMAT"" %
%   T4:23/DN  TEST_VP  "Povoleny cas najeti do vychozi polohy" %
%   N7:75/12  POMOC23 %
%   N7:75/11  POMOC22 %
% Rung: 13 %
SOR XIO N7:75/11 JMP Q7:1 EOR
%   N7:75/11  POMOC22 %
% Rung: 14 %
SOR XIO I:2.0/2 OTL N7:46/6 EOR
%   I:2.0/2  OZ  "Oddelovani parizonu zasunuto" %
%   N7:46/6  ERROR_OZ  "Oddelovani parizonu se nezasunulo" %
% Rung: 15 %
SOR XIC N7:8/9 XIO I:2.1/8 OTL N7:46/13 EOR
%   N7:8/9  _HLAVA  "Potvrzena predvolba" %
%   I:2.1/8  HN  "Ztracena hlava nahore" %
%   N7:46/13  ERROR_HN  "Ztracena hlava nebyla nahore" %
% Rung: 16 %
SOR XIC N7:8/12 BST XIO I:2.1/6 OTL N7:47/3 NXB XIO I:2.1/4 OTL N7:47/2 BND EOR
%   N7:8/12  _STABILIZ  "Potvrzena predvolba" %
%   I:2.1/6  STN  "Stabiliz. trn nahore" %
%   N7:47/3  ERROR_STN  "Stabiliz. trn nebyl nahore" %
%   I:2.1/4  SMO  "Stabiliz. maska otevrena" %
%   N7:47/2  ERROR_SMO  "Stabiliz. maska nebyla otevrena" %

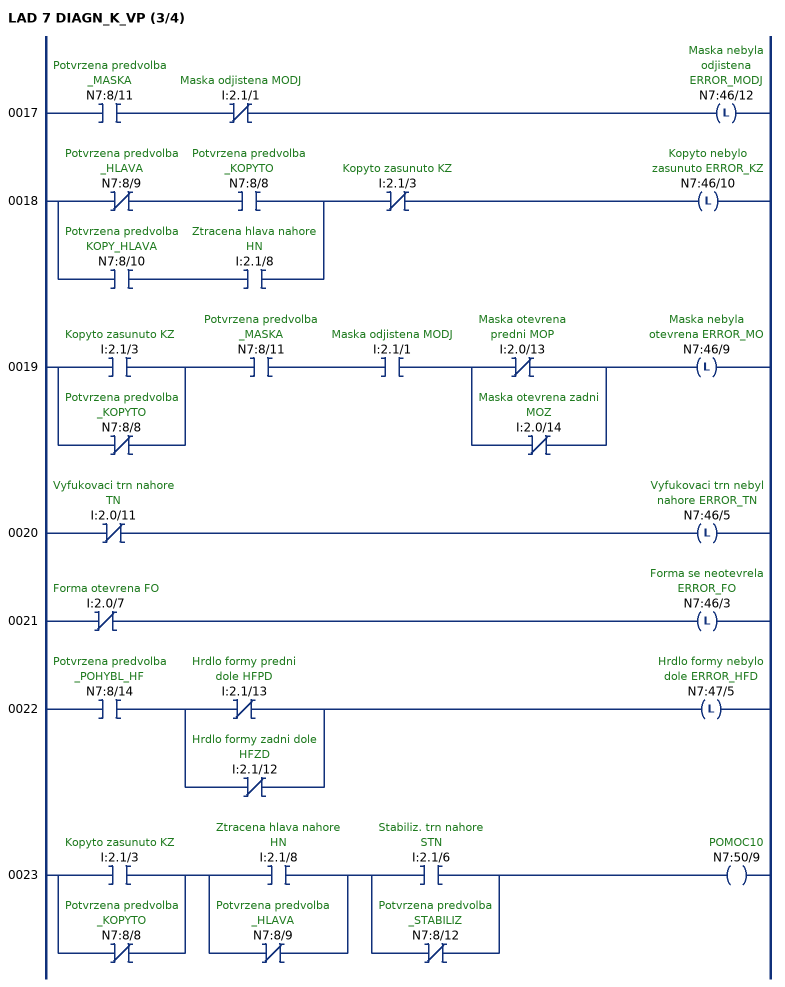
% Rung: 17 %
SOR XIC N7:8/11 XIO I:2.1/1 OTL N7:46/12 EOR
%   N7:8/11  _MASKA  "Potvrzena predvolba" %
%   I:2.1/1  MODJ  "Maska odjistena" %
%   N7:46/12  ERROR_MODJ  "Maska nebyla odjistena" %
% Rung: 18 %
SOR BST XIO N7:8/9 XIC N7:8/8 NXB XIC N7:8/10 XIC I:2.1/8 BND XIO I:2.1/3 OTL N7:46/10 EOR
%   N7:8/9  _HLAVA  "Potvrzena predvolba" %
%   N7:8/8  _KOPYTO  "Potvrzena predvolba" %
%   N7:8/10  KOPY_HLAVA  "Potvrzena predvolba" %
%   I:2.1/8  HN  "Ztracena hlava nahore" %
%   I:2.1/3  KZ  "Kopyto zasunuto" %
%   N7:46/10  ERROR_KZ  "Kopyto nebylo zasunuto" %
% Rung: 19 %
SOR BST XIC I:2.1/3 NXB XIO N7:8/8 BND XIC N7:8/11 XIC I:2.1/1 BST XIO I:2.0/13 NXB XIO I:2.0/14 BND OTL N7:46/9 EOR
%   I:2.1/3  KZ  "Kopyto zasunuto" %
%   N7:8/8  _KOPYTO  "Potvrzena predvolba" %
%   N7:8/11  _MASKA  "Potvrzena predvolba" %
%   I:2.1/1  MODJ  "Maska odjistena" %
%   I:2.0/13  MOP  "Maska otevrena predni" %
%   I:2.0/14  MOZ  "Maska otevrena zadni" %
%   N7:46/9  ERROR_MO  "Maska nebyla otevrena" %
% Rung: 20 %
SOR XIO I:2.0/11 OTL N7:46/5 EOR
%   I:2.0/11  TN  "Vyfukovaci trn nahore" %
%   N7:46/5  ERROR_TN  "Vyfukovaci trn nebyl nahore" %
% Rung: 21 %
SOR XIO I:2.0/7 OTL N7:46/3 EOR
%   I:2.0/7  FO  "Forma otevrena" %
%   N7:46/3  ERROR_FO  "Forma se neotevrela" %
% Rung: 22 %
SOR XIC N7:8/14 BST XIO I:2.1/13 NXB XIO I:2.1/12 BND OTL N7:47/5 EOR
%   N7:8/14  _POHYBL_HF  "Potvrzena predvolba" %
%   I:2.1/13  HFPD  "Hrdlo formy predni dole" %
%   I:2.1/12  HFZD  "Hrdlo formy zadni dole" %
%   N7:47/5  ERROR_HFD  "Hrdlo formy nebylo dole" %
% Rung: 23 %
SOR BST XIC I:2.1/3 NXB XIO N7:8/8 BND BST XIC I:2.1/8 NXB XIO N7:8/9 BND BST XIC I:2.1/6 NXB XIO N7:8/12 BND OTE N7:50/9 EOR
%   I:2.1/3  KZ  "Kopyto zasunuto" %
%   N7:8/8  _KOPYTO  "Potvrzena predvolba" %
%   I:2.1/8  HN  "Ztracena hlava nahore" %
%   N7:8/9  _HLAVA  "Potvrzena predvolba" %
%   I:2.1/6  STN  "Stabiliz. trn nahore" %
%   N7:8/12  _STABILIZ  "Potvrzena predvolba" %
%   N7:50/9  POMOC10 %

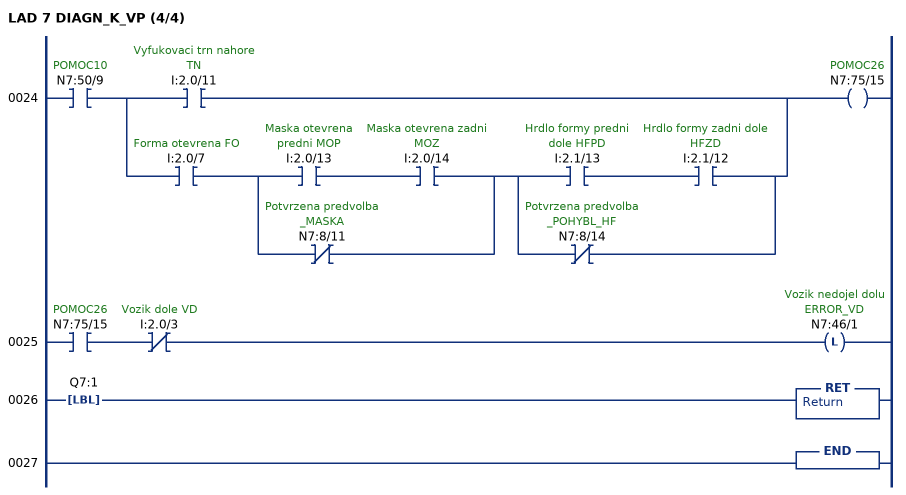
% Rung: 24 %
SOR XIC N7:50/9 BST XIC I:2.0/11 NXB XIC I:2.0/7 BST XIC I:2.0/13 XIC I:2.0/14 NXB XIO N7:8/11 BND BST XIC I:2.1/13 XIC I:2.1/12 NXB XIO N7:8/14 BND BND OTE N7:75/15 EOR
%   N7:50/9  POMOC10 %
%   I:2.0/11  TN  "Vyfukovaci trn nahore" %
%   I:2.0/7  FO  "Forma otevrena" %
%   I:2.0/13  MOP  "Maska otevrena predni" %
%   I:2.0/14  MOZ  "Maska otevrena zadni" %
%   N7:8/11  _MASKA  "Potvrzena predvolba" %
%   I:2.1/13  HFPD  "Hrdlo formy predni dole" %
%   I:2.1/12  HFZD  "Hrdlo formy zadni dole" %
%   N7:8/14  _POHYBL_HF  "Potvrzena predvolba" %
%   N7:75/15  POMOC26 %
% Rung: 25 %
SOR XIC N7:75/15 XIO I:2.0/3 OTL N7:46/1 EOR
%   N7:75/15  POMOC26 %
%   I:2.0/3  VD  "Vozik dole" %
%   N7:46/1  ERROR_VD  "Vozik nedojel dolu" %
% Rung: 26 %
SOR LBL Q7:1 RET EOR
% Rung: 27 %
SOR END EOR

LADDER 8 "HYDR_AGREG"
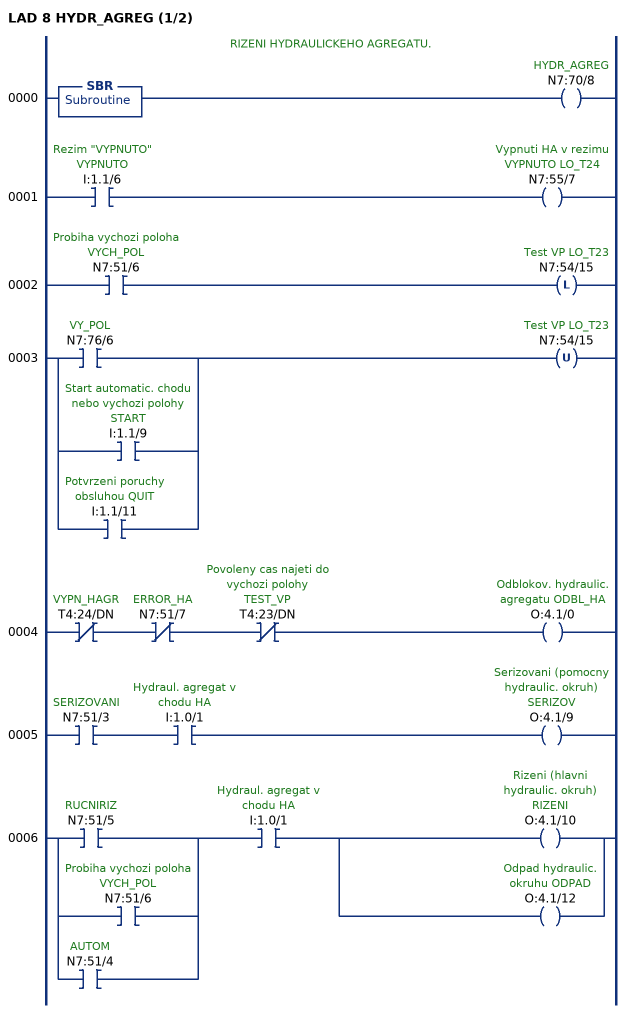
% Rung: 0 %
% RIZENI HYDRAULICKEHO AGREGATU. %
SOR SBR OTE N7:70/8 EOR
%   N7:70/8  HYDR_AGREG %
% Rung: 1 %
SOR XIC I:1.1/6 OTE N7:55/7 EOR
%   I:1.1/6  VYPNUTO  "Rezim "VYPNUTO"" %
%   N7:55/7  LO_T24  "Vypnuti HA v rezimu VYPNUTO" %
% Rung: 2 %
SOR XIC N7:51/6 OTL N7:54/15 EOR
%   N7:51/6  VYCH_POL  "Probiha vychozi poloha" %
%   N7:54/15  LO_T23  "Test VP" %
% Rung: 3 %
SOR BST XIC N7:76/6 NXB XIC I:1.1/9 NXB XIC I:1.1/11 BND OTU N7:54/15 EOR
%   N7:76/6  VY_POL %
%   I:1.1/9  START  "Start automatic. chodu nebo vychozi polohy" %
%   I:1.1/11  QUIT  "Potvrzeni poruchy obsluhou" %
%   N7:54/15  LO_T23  "Test VP" %
% Rung: 4 %
SOR XIO T4:24/DN XIO N7:51/7 XIO T4:23/DN OTE O:4.1/0 EOR
%   T4:24/DN  VYPN_HAGR %
%   N7:51/7  ERROR_HA %
%   T4:23/DN  TEST_VP  "Povoleny cas najeti do vychozi polohy" %
%   O:4.1/0  ODBL_HA  "Odblokov. hydraulic. agregatu" %
% Rung: 5 %
SOR XIC N7:51/3 XIC I:1.0/1 OTE O:4.1/9 EOR
%   N7:51/3  SERIZOVANI %
%   I:1.0/1  HA  "Hydraul. agregat v chodu" %
%   O:4.1/9  SERIZOV  "Serizovani (pomocny hydraulic. okruh)" %
% Rung: 6 %
SOR BST XIC N7:51/5 NXB XIC N7:51/6 NXB XIC N7:51/4 BND XIC I:1.0/1 BST OTE O:4.1/10 NXB OTE O:4.1/12 BND EOR
%   N7:51/5  RUCNIRIZ %
%   N7:51/6  VYCH_POL  "Probiha vychozi poloha" %
%   N7:51/4  AUTOM %
%   I:1.0/1  HA  "Hydraul. agregat v chodu" %
%   O:4.1/10  RIZENI  "Rizeni (hlavni hydraulic. okruh)" %
%   O:4.1/12  ODPAD  "Odpad hydraulic. okruhu" %

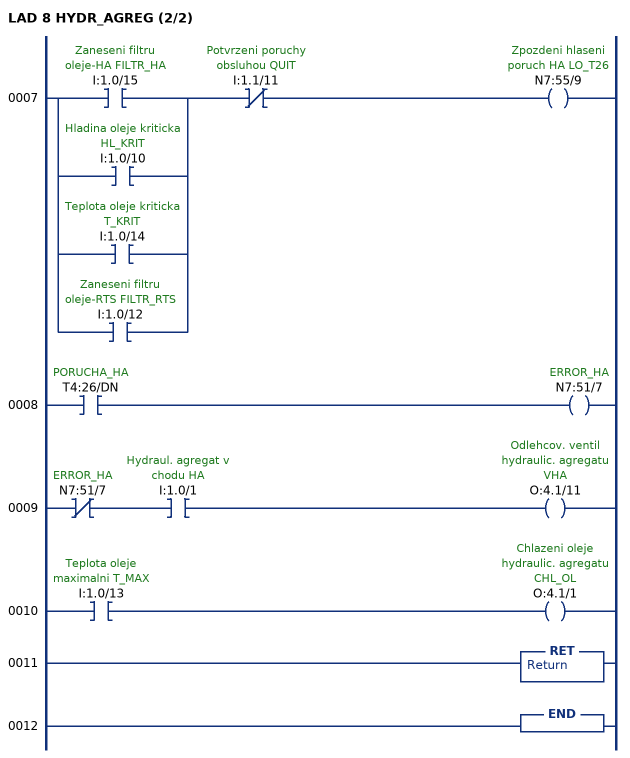
% Rung: 7 %
SOR BST XIC I:1.0/15 NXB XIC I:1.0/10 NXB XIC I:1.0/14 NXB XIC I:1.0/12 BND XIO I:1.1/11 OTE N7:55/9 EOR
%   I:1.0/15  FILTR_HA  "Zaneseni filtru oleje-HA" %
%   I:1.0/10  HL_KRIT  "Hladina oleje kriticka" %
%   I:1.0/14  T_KRIT  "Teplota oleje kriticka" %
%   I:1.0/12  FILTR_RTS  "Zaneseni filtru oleje-RTS" %
%   I:1.1/11  QUIT  "Potvrzeni poruchy obsluhou" %
%   N7:55/9  LO_T26  "Zpozdeni hlaseni poruch HA" %
% Rung: 8 %
SOR XIC T4:26/DN OTE N7:51/7 EOR
%   T4:26/DN  PORUCHA_HA %
%   N7:51/7  ERROR_HA %
% Rung: 9 %
SOR XIO N7:51/7 XIC I:1.0/1 OTE O:4.1/11 EOR
%   N7:51/7  ERROR_HA %
%   I:1.0/1  HA  "Hydraul. agregat v chodu" %
%   O:4.1/11  VHA  "Odlehcov. ventil hydraulic. agregatu" %
% Rung: 10 %
SOR XIC I:1.0/13 OTE O:4.1/1 EOR
%   I:1.0/13  T_MAX  "Teplota oleje maximalni" %
%   O:4.1/1  CHL_OL  "Chlazeni oleje hydraulic. agregatu" %
% Rung: 11 %
SOR RET EOR
% Rung: 12 %
SOR END EOR

LADDER 9 "VODA_POHON"
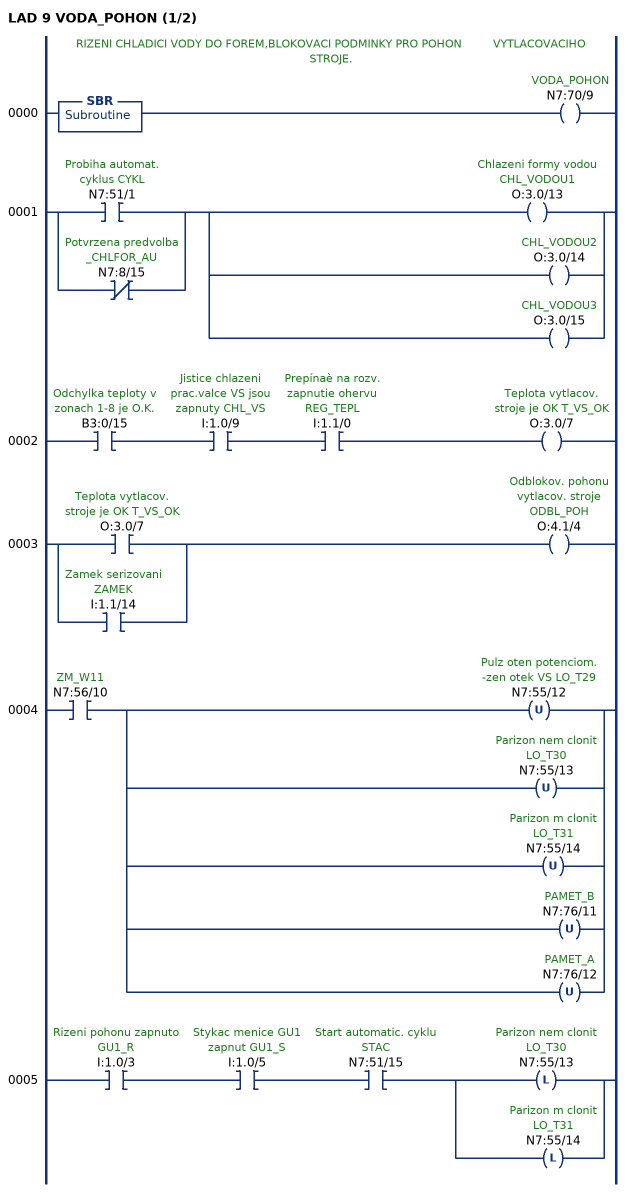
% Rung: 0 %
% RIZENI CHLADICI VODY DO FOREM,BLOKOVACI PODMINKY PRO POHON         VYTLACOVACIHO STROJE. %
SOR SBR OTE N7:70/9 EOR
%   N7:70/9  VODA_POHON %
% Rung: 1 %
SOR BST XIC N7:51/1 NXB XIO N7:8/15 BND BST OTE O:3.0/13 NXB OTE O:3.0/14 NXB OTE O:3.0/15 BND EOR
%   N7:51/1  CYKL  "Probiha automat. cyklus" %
%   N7:8/15  _CHLFOR_AU  "Potvrzena predvolba" %
%   O:3.0/13  CHL_VODOU1  "Chlazeni formy vodou" %
%   O:3.0/14  CHL_VODOU2 %
%   O:3.0/15  CHL_VODOU3 %
% Rung: 2 %
SOR XIC B3:0/15 XIC I:1.0/9 XIC I:1.1/0 OTE O:3.0/7 EOR
%   B3:0/15  "Odchylka teploty v zonach 1-8 je O.K." %
%   I:1.0/9  CHL_VS  "Jistice chlazeni prac.valce VS jsou zapnuty" %
%   I:1.1/0  REG_TEPL  "Prepínaè na rozv. zapnutie ohervu" %
%   O:3.0/7  T_VS_OK  "Teplota vytlacov. stroje je OK" %
% Rung: 3 %
SOR BST XIC O:3.0/7 NXB XIC I:1.1/14 BND OTE O:4.1/4 EOR
%   O:3.0/7  T_VS_OK  "Teplota vytlacov. stroje je OK" %
%   I:1.1/14  ZAMEK  "Zamek serizovani" %
%   O:4.1/4  ODBL_POH  "Odblokov. pohonu vytlacov. stroje" %
% Rung: 4 %
SOR XIC N7:56/10 BST OTU N7:55/12 NXB OTU N7:55/13 NXB OTU N7:55/14 NXB OTU N7:76/11 NXB OTU N7:76/12 BND EOR
%   N7:56/10  ZM_W11 %
%   N7:55/12  LO_T29  "Pulz oten potenciom. -zen otek VS" %
%   N7:55/13  LO_T30  "Parizon nem clonit" %
%   N7:55/14  LO_T31  "Parizon m clonit" %
%   N7:76/11  PAMET_B %
%   N7:76/12  PAMET_A %
% Rung: 5 %
SOR XIC I:1.0/3 XIC I:1.0/5 XIC N7:51/15 BST OTL N7:55/13 NXB OTL N7:55/14 BND EOR
%   I:1.0/3  GU1_R  "Rizeni pohonu zapnuto" %
%   I:1.0/5  GU1_S  "Stykac menice GU1 zapnut" %
%   N7:51/15  STAC  "Start automatic. cyklu" %
%   N7:55/13  LO_T30  "Parizon nem clonit" %
%   N7:55/14  LO_T31  "Parizon m clonit" %

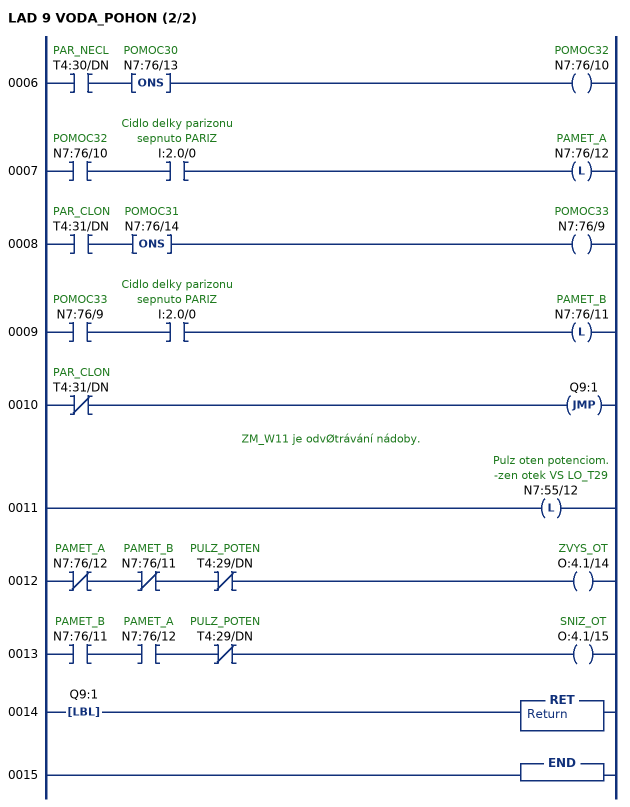
% Rung: 6 %
SOR XIC T4:30/DN OSR N7:76/13 OTE N7:76/10 EOR
%   T4:30/DN  PAR_NECL %
%   N7:76/13  POMOC30 %
%   N7:76/10  POMOC32 %
% Rung: 7 %
SOR XIC N7:76/10 XIC I:2.0/0 OTL N7:76/12 EOR
%   N7:76/10  POMOC32 %
%   I:2.0/0  PARIZ  "Cidlo delky parizonu sepnuto" %
%   N7:76/12  PAMET_A %
% Rung: 8 %
SOR XIC T4:31/DN OSR N7:76/14 OTE N7:76/9 EOR
%   T4:31/DN  PAR_CLON %
%   N7:76/14  POMOC31 %
%   N7:76/9  POMOC33 %
% Rung: 9 %
SOR XIC N7:76/9 XIC I:2.0/0 OTL N7:76/11 EOR
%   N7:76/9  POMOC33 %
%   I:2.0/0  PARIZ  "Cidlo delky parizonu sepnuto" %
%   N7:76/11  PAMET_B %
% Rung: 10 %
SOR XIO T4:31/DN JMP Q9:1 EOR
%   T4:31/DN  PAR_CLON %
% Rung: 11 %
% ZM_W11 je odvØtrávání nádoby. %
SOR OTL N7:55/12 EOR
%   N7:55/12  LO_T29  "Pulz oten potenciom. -zen otek VS" %
% Rung: 12 %
SOR XIO N7:76/12 XIO N7:76/11 XIO T4:29/DN OTE O:4.1/14 EOR
%   N7:76/12  PAMET_A %
%   N7:76/11  PAMET_B %
%   T4:29/DN  PULZ_POTEN %
%   O:4.1/14  ZVYS_OT %
% Rung: 13 %
SOR XIC N7:76/11 XIC N7:76/12 XIO T4:29/DN OTE O:4.1/15 EOR
%   N7:76/11  PAMET_B %
%   N7:76/12  PAMET_A %
%   T4:29/DN  PULZ_POTEN %
%   O:4.1/15  SNIZ_OT %
% Rung: 14 %
SOR LBL Q9:1 RET EOR
% Rung: 15 %
SOR END EOR

LADDER 10 "REZIM_SER"
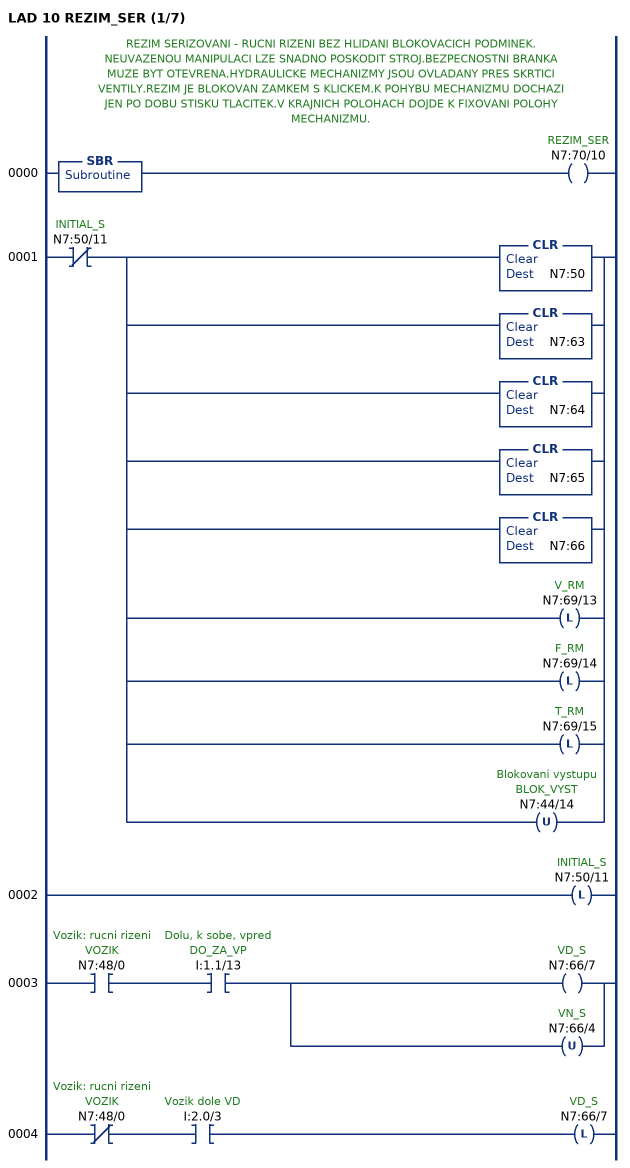
% Rung: 0 %
% REZIM SERIZOVANI - RUCNI RIZENI BEZ HLIDANI BLOKOVACICH PODMINEK.
% NEUVAZENOU MANIPULACI LZE SNADNO POSKODIT STROJ.BEZPECNOSTNI BRANKA
% MUZE BYT OTEVRENA.HYDRAULICKE MECHANIZMY JSOU OVLADANY PRES SKRTICI
% VENTILY.REZIM JE BLOKOVAN ZAMKEM S KLICKEM.K POHYBU MECHANIZMU DOCHAZI
% JEN PO DOBU STISKU TLACITEK.V KRAJNICH POLOHACH DOJDE K FIXOVANI POLOHY
% MECHANIZMU. %
SOR SBR OTE N7:70/10 EOR
%   N7:70/10  REZIM_SER %
% Rung: 1 %
SOR XIO N7:50/11 BST CLR N7:50 NXB CLR N7:63 NXB CLR N7:64 NXB CLR N7:65 NXB CLR N7:66 NXB OTL N7:69/13 NXB OTL N7:69/14 NXB OTL N7:69/15 NXB OTU N7:44/14 BND EOR
%   N7:50/11  INITIAL_S %
%   CLR N7:50  "Pomocne merkry" %
%   CLR N7:63  "Merkry vystupu rucniho rezimu" %
%   CLR N7:64  "Merkry vystupu rucniho rezimu" %
%   CLR N7:65  "Merkry vystupu rezimu serizovani" %
%   CLR N7:66  "Merkry vystupu rezimu serizovani" %
%   N7:69/13  V_RM %
%   N7:69/14  F_RM %
%   N7:69/15  T_RM %
%   N7:44/14  BLOK_VYST  "Blokovani vystupu" %
% Rung: 2 %
SOR OTL N7:50/11 EOR
%   N7:50/11  INITIAL_S %
% Rung: 3 %
SOR XIC N7:48/0 XIC I:1.1/13 BST OTE N7:66/7 NXB OTU N7:66/4 BND EOR
%   N7:48/0  VOZIK  "Vozik: rucni rizeni" %
%   I:1.1/13  DO_ZA_VP  "Dolu, k sobe, vpred" %
%   N7:66/7  VD_S %
%   N7:66/4  VN_S %
% Rung: 4 %
SOR XIO N7:48/0 XIC I:2.0/3 OTL N7:66/7 EOR
%   N7:48/0  VOZIK  "Vozik: rucni rizeni" %
%   I:2.0/3  VD  "Vozik dole" %
%   N7:66/7  VD_S %

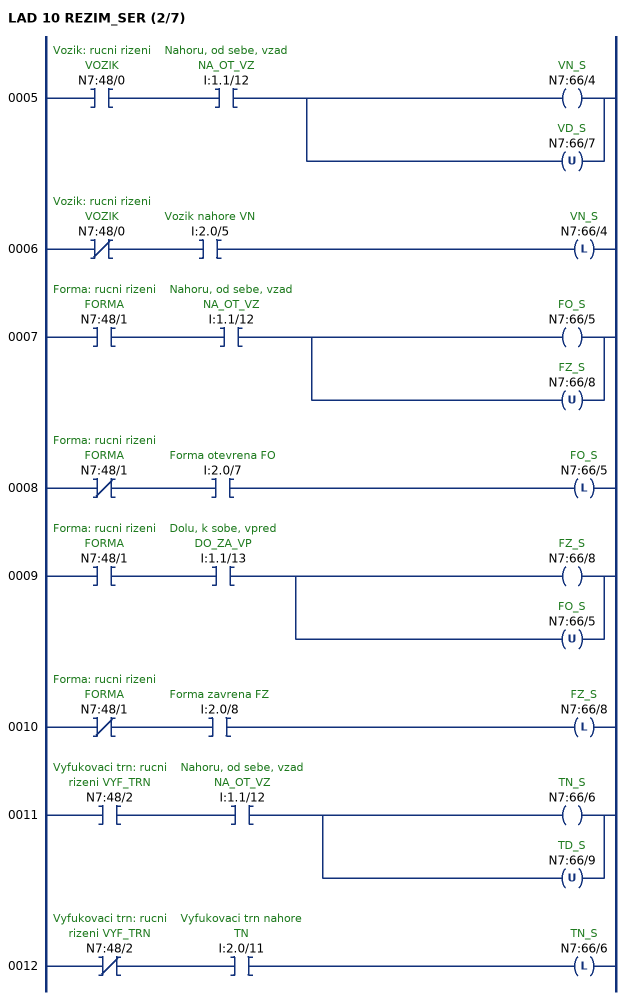
% Rung: 5 %
SOR XIC N7:48/0 XIC I:1.1/12 BST OTE N7:66/4 NXB OTU N7:66/7 BND EOR
%   N7:48/0  VOZIK  "Vozik: rucni rizeni" %
%   I:1.1/12  NA_OT_VZ  "Nahoru, od sebe, vzad" %
%   N7:66/4  VN_S %
%   N7:66/7  VD_S %
% Rung: 6 %
SOR XIO N7:48/0 XIC I:2.0/5 OTL N7:66/4 EOR
%   N7:48/0  VOZIK  "Vozik: rucni rizeni" %
%   I:2.0/5  VN  "Vozik nahore" %
%   N7:66/4  VN_S %
% Rung: 7 %
SOR XIC N7:48/1 XIC I:1.1/12 BST OTE N7:66/5 NXB OTU N7:66/8 BND EOR
%   N7:48/1  FORMA  "Forma: rucni rizeni" %
%   I:1.1/12  NA_OT_VZ  "Nahoru, od sebe, vzad" %
%   N7:66/5  FO_S %
%   N7:66/8  FZ_S %
% Rung: 8 %
SOR XIO N7:48/1 XIC I:2.0/7 OTL N7:66/5 EOR
%   N7:48/1  FORMA  "Forma: rucni rizeni" %
%   I:2.0/7  FO  "Forma otevrena" %
%   N7:66/5  FO_S %
% Rung: 9 %
SOR XIC N7:48/1 XIC I:1.1/13 BST OTE N7:66/8 NXB OTU N7:66/5 BND EOR
%   N7:48/1  FORMA  "Forma: rucni rizeni" %
%   I:1.1/13  DO_ZA_VP  "Dolu, k sobe, vpred" %
%   N7:66/8  FZ_S %
%   N7:66/5  FO_S %
% Rung: 10 %
SOR XIO N7:48/1 XIC I:2.0/8 OTL N7:66/8 EOR
%   N7:48/1  FORMA  "Forma: rucni rizeni" %
%   I:2.0/8  FZ  "Forma zavrena" %
%   N7:66/8  FZ_S %
% Rung: 11 %
SOR XIC N7:48/2 XIC I:1.1/12 BST OTE N7:66/6 NXB OTU N7:66/9 BND EOR
%   N7:48/2  VYF_TRN  "Vyfukovaci trn: rucni rizeni" %
%   I:1.1/12  NA_OT_VZ  "Nahoru, od sebe, vzad" %
%   N7:66/6  TN_S %
%   N7:66/9  TD_S %
% Rung: 12 %
SOR XIO N7:48/2 XIC I:2.0/11 OTL N7:66/6 EOR
%   N7:48/2  VYF_TRN  "Vyfukovaci trn: rucni rizeni" %
%   I:2.0/11  TN  "Vyfukovaci trn nahore" %
%   N7:66/6  TN_S %

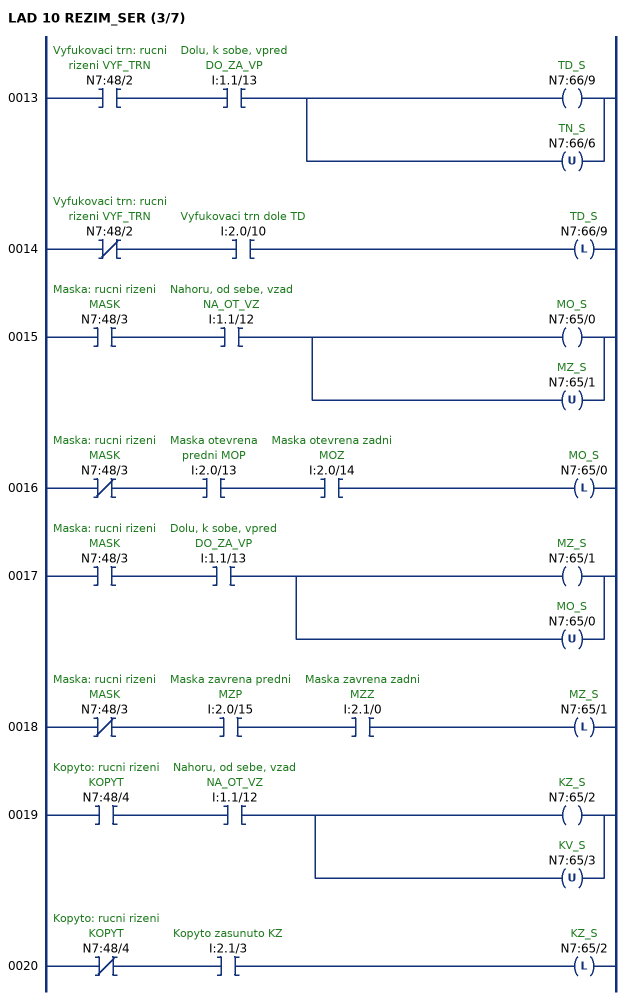
% Rung: 13 %
SOR XIC N7:48/2 XIC I:1.1/13 BST OTE N7:66/9 NXB OTU N7:66/6 BND EOR
%   N7:48/2  VYF_TRN  "Vyfukovaci trn: rucni rizeni" %
%   I:1.1/13  DO_ZA_VP  "Dolu, k sobe, vpred" %
%   N7:66/9  TD_S %
%   N7:66/6  TN_S %
% Rung: 14 %
SOR XIO N7:48/2 XIC I:2.0/10 OTL N7:66/9 EOR
%   N7:48/2  VYF_TRN  "Vyfukovaci trn: rucni rizeni" %
%   I:2.0/10  TD  "Vyfukovaci trn dole" %
%   N7:66/9  TD_S %
% Rung: 15 %
SOR XIC N7:48/3 XIC I:1.1/12 BST OTE N7:65/0 NXB OTU N7:65/1 BND EOR
%   N7:48/3  MASK  "Maska: rucni rizeni" %
%   I:1.1/12  NA_OT_VZ  "Nahoru, od sebe, vzad" %
%   N7:65/0  MO_S %
%   N7:65/1  MZ_S %
% Rung: 16 %
SOR XIO N7:48/3 XIC I:2.0/13 XIC I:2.0/14 OTL N7:65/0 EOR
%   N7:48/3  MASK  "Maska: rucni rizeni" %
%   I:2.0/13  MOP  "Maska otevrena predni" %
%   I:2.0/14  MOZ  "Maska otevrena zadni" %
%   N7:65/0  MO_S %
% Rung: 17 %
SOR XIC N7:48/3 XIC I:1.1/13 BST OTE N7:65/1 NXB OTU N7:65/0 BND EOR
%   N7:48/3  MASK  "Maska: rucni rizeni" %
%   I:1.1/13  DO_ZA_VP  "Dolu, k sobe, vpred" %
%   N7:65/1  MZ_S %
%   N7:65/0  MO_S %
% Rung: 18 %
SOR XIO N7:48/3 XIC I:2.0/15 XIC I:2.1/0 OTL N7:65/1 EOR
%   N7:48/3  MASK  "Maska: rucni rizeni" %
%   I:2.0/15  MZP  "Maska zavrena predni" %
%   I:2.1/0  MZZ  "Maska zavrena zadni" %
%   N7:65/1  MZ_S %
% Rung: 19 %
SOR XIC N7:48/4 XIC I:1.1/12 BST OTE N7:65/2 NXB OTU N7:65/3 BND EOR
%   N7:48/4  KOPYT  "Kopyto: rucni rizeni" %
%   I:1.1/12  NA_OT_VZ  "Nahoru, od sebe, vzad" %
%   N7:65/2  KZ_S %
%   N7:65/3  KV_S %
% Rung: 20 %
SOR XIO N7:48/4 XIC I:2.1/3 OTL N7:65/2 EOR
%   N7:48/4  KOPYT  "Kopyto: rucni rizeni" %
%   I:2.1/3  KZ  "Kopyto zasunuto" %
%   N7:65/2  KZ_S %

